FUNCTION_BLOCK "Epever_solar_charge_controller"   // FB109, SCL
{ S7_Optimized_Access := 'TRUE' }
VERSION : 0.1
   VAR_INPUT
      mb_addr : UInt := 1;
      on : Bool;
   END_VAR
   VAR_OUTPUT
      PV_array_input_voltage : Real;
      PV_array_input_current : Real;
      PV_array_input_power : Real;
      battery_power : Real;
      load_voltage : Real;
      load_current : Real;
      load_power : Real;
      battery_temperature : Real;
      temperature_inside_equipment : Real;
      battery_soc : Real;   // The percentage of battery's remaining capacity
      remote_battery_temperature : Real;
      battery_real_rated_power : Real;
      _ : Bool;
      PV_voltage_today_Maximum : Real;
      PV_voltage_today_Minimum : Real;
      Battery_voltage_today_Maximum : Real;
      Battery_voltage_today_Minimum : Real;
      Consumed_energy_today : Real;
      Consumed_energy_this_month : Real;
      Consumed_energy_this_year : Real;
      Consumed_energy_total : Real;
      Generated_energy_today : Real;
      Generated_energy_this_month : Real;
      Generated_energy_this_year : Real;
      Generated_energy_total : Real;
      Battery_voltage : Real;
      Battery_current : Real;
      __ : Bool;
      charging_status : Struct
         No_charging : Bool;
         Float : Bool;
         Boost : Bool;
         Equalization : Bool;
      END_STRUCT;
   END_VAR
   VAR_IN_OUT
      mb_query : "mb_query";
   END_VAR
   VAR
      sb : "mb_station_block_udt";
      read3 : Struct
         load_short : Bool;   // [08]
         load_over_current : Bool;   // [09]
         Input_is_over_current : Bool;   // [10]
         Anti_reverse_MOSFET_is_short : Bool;   // [11]
         Charging_or_Anti_reverse_MOSFET_is_short : Bool;   // [12]
         Charging_MOSFET_is_short : Bool;   // [13]
         x14 : Bool;   // [14]
         x15 : Bool;   // [15]
         Running : Bool;   // [00] - Standby
         Normal : Bool;   // [01] - Fault
         charging_status_0 : Bool;   // [02]
         charging_status_1 : Bool;   // [03]
         PV_Input_is_short : Bool;   // [04]
         x05 : Bool;   // [05]
         x06 : Bool;   // [06]
         Load_MOSFET_is_short : Bool;   // [07]
      END_STRUCT;
      first_scan : Bool := true;
   END_VAR
   VAR_TEMP
      read1 : Struct
         PV_array_input_voltage : UInt;   // [3100]
         PV_array_input_current : UInt;   // [3101]
         PV_array_input_power : UDInt;   // [3102]
         z_1 : Array[1..3] of Word;
         battery_power : UDInt;   // [3106]
         z_2 : Array[1..4] of Word;
         load_voltage : UInt;   // [310C]
         load_current : UInt;   // [310D]
         load_power : UDInt;   // [310E]
         battery_temperature : UInt;   // [3110]
         temperature_inside_equipment : UInt;   // [3111]
         battery_soc : UInt;   // [311A] The percentage of battery's remaining capacity
         remote_battery_temperature : UInt;   // [311B]
         z_3 : UInt;
         battery_real_rated_power : UInt;   // [311D]
      END_STRUCT;
      read2 : Struct
         PV_voltage_today_Maximum : UInt;   // [3300]
         PV_voltage_today_Minimum : UInt;   // [3301]
         Battery_voltage_today_Maximum : UInt;   // [3302]
         Battery_voltage_today_Minimum : UInt;   // [3303]
         Consumed_energy_today : UDInt;   // [3304]
         Consumed_energy_this_month : UDInt;   // [3306]
         Consumed_energy_this_year : UDInt;   // [3308]
         Consumed_energy_total : UDInt;   // [330A]
         Generated_energy_today : UDInt;   // [330C]
         Generated_energy_this_month : UDInt;   // [330E]
         Generated_energy_this_year : UDInt;   // [3310]
         Generated_energy_total : UDInt;   // [3312]
         Battery_voltage : UInt;   // [331A]
         Battery_current : UDInt;   // [331B]
      END_STRUCT;
      tmp : Byte;
   END_VAR
BEGIN
   // Epever - solar charge controller 
   // v2.3 - 12 june 2015
   // 

   IF #first_scan THEN
       #sb.conf.read_only := true;
   END_IF;

   "mb_station_block_header"(sb := #sb, mb_query := #mb_query);
   #mb_query.mb_addr := #mb_addr; 

   #mb_query.mode := #mb_query.c.read.input_reg;
   #mb_query(data_addr := 16#3100, data_ptr := #read1);
   IF #mb_query.Done THEN
       #PV_array_input_voltage := UINT_TO_REAL(#read1.PV_array_input_voltage) / 100;
       #PV_array_input_current := UINT_TO_REAL(#read1.PV_array_input_current) / 100;
       #PV_array_input_power := UDINT_TO_REAL(ROR(IN := #read1.PV_array_input_power, N := 16)) / 100;
       #battery_power := UDINT_TO_REAL(ROR(IN := #read1.battery_power, N := 16)) / 100;
       #load_voltage := UINT_TO_REAL(#read1.load_voltage) / 100;
       #load_current := UINT_TO_REAL(#read1.load_current) / 100;
       #load_power := UDINT_TO_REAL(ROR(IN := #read1.load_power, N := 16)) / 100;
       #battery_temperature := UINT_TO_REAL(#read1.battery_temperature) / 100;
       #temperature_inside_equipment := UINT_TO_REAL(#read1.temperature_inside_equipment) / 100;
       #battery_soc := UINT_TO_REAL(#read1.battery_soc) / 100;
       #remote_battery_temperature := UINT_TO_REAL(#read1.remote_battery_temperature) / 100;
       #battery_real_rated_power := UINT_TO_REAL(#read1.battery_real_rated_power) / 100;
   END_IF;

   #mb_query(data_addr := 16#3300, data_ptr := #read2);
   IF #mb_query.Done THEN
       #PV_voltage_today_Maximum := UINT_TO_REAL(#read2.PV_voltage_today_Maximum) / 100;
       #PV_voltage_today_Minimum := UINT_TO_REAL(#read2.PV_voltage_today_Minimum) / 100;
       #Battery_voltage_today_Maximum := UINT_TO_REAL(#read2.Battery_voltage_today_Maximum) / 100;
       #Battery_voltage_today_Minimum := UINT_TO_REAL(#read2.Battery_voltage_today_Minimum) / 100;
       #Consumed_energy_today := UDINT_TO_REAL(ROR(IN := #read2.Consumed_energy_today, N := 16)) / 100;
       #Consumed_energy_this_month := UDINT_TO_REAL(ROR(IN := #read2.Consumed_energy_this_month, N := 16)) / 100;
       #Consumed_energy_this_year := UDINT_TO_REAL(ROR(IN := #read2.Consumed_energy_this_year, N := 16)) / 100;
       #Consumed_energy_total := UDINT_TO_REAL(ROR(IN := #read2.Consumed_energy_total, N := 16)) / 100;
       #Generated_energy_today := UDINT_TO_REAL(ROR(IN := #read2.Generated_energy_today, N := 16)) / 100;
       #Generated_energy_this_month := UDINT_TO_REAL(ROR(IN := #read2.Generated_energy_this_month, N := 16)) / 100;
       #Generated_energy_this_year := UDINT_TO_REAL(ROR(IN := #read2.Generated_energy_this_year, N := 16)) / 100;
       #Generated_energy_total := UDINT_TO_REAL(ROR(IN := #read2.Generated_energy_total, N := 16)) / 100;
       #Battery_voltage := UDINT_TO_REAL(#read2.Battery_voltage) / 100;
       #Battery_current := UDINT_TO_REAL(ROR(IN := #read2.Battery_current, N := 16)) / 100;
   END_IF;


   #mb_query(data_addr := 16#3201, data_ptr := #read3);
   #tmp.%X0 := #read3.charging_status_0;
   #tmp.%X1 := #read3.charging_status_1;
   #charging_status.No_charging := #tmp = 0;
   #charging_status.Float := #tmp = 1;
   #charging_status.Boost := #tmp = 2;
   #charging_status.Equalization := #tmp = 3;

   #mb_query.mode := #mb_query.c.write.single_discrete_output;
   #tmp.%X0 := #on;
   #mb_query(data_addr := 0, data_ptr := #tmp);

   "mb_station_block_footer"(sb := #sb, mb_query := #mb_query);


   (*
   - 16bit MODBUS addresses (per the modbus.org spec)
   - BPS: 115200 baud
   - Parity: None
   - Data bits: 8
   - Stop bits: 1
   - Flow control: None

   Pin definition RJ45 
   1   Power supply output +7.5
   2   Power supply output +7.5
   3   RS-485 - A
   4   RS-485 - A
   5   RS-485 - B
   6   RS-485 - B
   7   Ground
   8   Ground

   *)
END_FUNCTION_BLOCK

// folder: Library/Modbus/Station blocks/sb Untested/F/Floridan

FUNCTION_BLOCK "Floridan_Uniflo_1200"   // FB83, SCL
{ S7_Optimized_Access := 'TRUE' }
VERSION : 0.1
   VAR_INPUT
      mb_addr : USInt;
      delay : Time := T#10S;
   END_VAR
   VAR_OUTPUT
      energi : LReal;   // [MJ]
      vol_measured : LReal;   // [m3]
      vol_conv : LReal;   // [Nm3]
      pressure : LReal;   // [bar A]
      temperature : LReal;
   END_VAR
   VAR_IN_OUT
      mb_query : "mb_query";
   END_VAR
   VAR
      sb : "mb_station_block_udt";
      battery_remaining : UInt;
      mb_delay : "mb_delay";
      serial_number : String[6];
   END_VAR
   VAR_TEMP
      dommy : Bool;
      c : Int;
      "dword" : DWord;
   END_VAR
BEGIN
   // Flonidan - Uniflo 1200 GVEC
   // Product number: 061864X-YYY
   //
   // - https://www.gavilar.nl/files/communicationboard230210_1521630740_b6a3b533.pdf
   // - M/06180XX/24

   "mb_station_block_header"(sb := #sb, mb_query := #mb_query);
   #mb_query.mb_addr := #mb_addr; // Device address.

   // Reduce power consumption, by halting execution. Nice if the device is running 
   // on battery. mb_delay is located inside the mb_extended_features.scl file.
   #mb_delay(delay := #delay, mb_query := #mb_query);

   #mb_query.mb_addr.%X5 := 0; // - Last bits of mb_addr is used for expanding 
   #mb_query.mb_addr.%X6 := 0; //   register addr, this means that only addr 1
   #mb_query.mb_addr.%X7 := 0; //   to 31 on the bus may be used.

   #mb_query.mode := #mb_query.c.read.holding_reg;

   #mb_query(data_addr := 123, data_ptr := #battery_remaining);
   #mb_query(data_addr := 2833, data_ptr := #serial_number); // Serial number 

   #mb_query.conf.buffer_handler := false;

   #mb_query(data_addr := 56, data_len := 44, data_ptr := #dommy);
   IF #mb_query.Done THEN
       #vol_conv := "intreal"(mb_query := #mb_query, addr := 16#70 / 2);
       #"dword".%B3 := #mb_query.z.buffer[16]; // 16#80/2=64, (64-56)*2=16
       #"dword".%B2 := #mb_query.z.buffer[17];
       #"dword".%B1 := #mb_query.z.buffer[18];
       #"dword".%B0 := #mb_query.z.buffer[19];
       #pressure := DWORD_TO_REAL(#"dword");
       #"dword".%B3 := #mb_query.z.buffer[20]; // 16#84/2=66, (66-56)*2=20
       #"dword".%B2 := #mb_query.z.buffer[21];
       #"dword".%B1 := #mb_query.z.buffer[22];
       #"dword".%B0 := #mb_query.z.buffer[23];
       #temperature := DWORD_TO_REAL(#"dword");
       #energi := "intreal"(mb_query := #mb_query, addr := 16#90 / 2);
       #vol_measured := "intreal"(mb_query := #mb_query, addr := 16#98 / 2);
   END_IF;

   #mb_query.data_len := #mb_query.c.auto_len;
   #mb_query.conf.buffer_handler := true;
   "mb_station_block_footer"(sb := #sb, mb_query := #mb_query);
END_FUNCTION_BLOCK

FUNCTION "intreal" : LReal   // FC16, SCL
{ S7_Optimized_Access := 'TRUE' }
VERSION : 0.1
   VAR_INPUT
      mb_query : "mb_query";
      addr : UInt;
   END_VAR
   VAR_TEMP
      dw : UDInt;
      r : DWord;
      bo : UDInt;
   END_VAR
BEGIN
   // Uniflo 1200 has a special datatype named
   // int-real, this block decode that data type.

   // buffer offset
   #bo := (#addr - #mb_query.data_addr) * 2;

   // The integer part of the value, little endian.
   #dw.%B3 := #mb_query.z.buffer[#bo + 0];
   #dw.%B2 := #mb_query.z.buffer[#bo + 1];
   #dw.%B1 := #mb_query.z.buffer[#bo + 2];
   #dw.%B0 := #mb_query.z.buffer[#bo + 3];
   #intreal := UDINT_TO_LREAL(#dw);

   // The decimal part of the value, little endian.
   // Stored as a real (IEEE754).
   #r.%B3 := #mb_query.z.buffer[#bo + 4];
   #r.%B2 := #mb_query.z.buffer[#bo + 5];
   #r.%B1 := #mb_query.z.buffer[#bo + 6];
   #r.%B0 := #mb_query.z.buffer[#bo + 7];
   #intreal += DWORD_TO_REAL(#r);
END_FUNCTION

// folder: Library/Modbus/Station blocks/sb Untested/G

FUNCTION_BLOCK "G_Instruments_GpH141_MB"   // FB26, SCL
{ S7_Optimized_Access := 'TRUE' }
VERSION : 0.1
   VAR_INPUT
      mb_addr : USInt;
   END_VAR
   VAR_OUTPUT
      voltage_mV : Real;
      pH : Real;
      temperature : Real;
   END_VAR
   VAR_IN_OUT
      mb_query : "mb_query";
   END_VAR
   VAR
      sb : "mb_station_block_udt";
      change_mb_addr : Struct
         old : UInt;
         new : UInt;
      END_STRUCT;
   END_VAR
   VAR_TEMP
      read1 : Struct
         voltage : Int;
         pH : Int;   // compensated for temperature
         temperature : Int;
      END_STRUCT;
   END_VAR
BEGIN
   // G Instruments - GpH141-MB - pH/ORP Transmitter
   // Part number: 30535.
   // http://www.ginstruments.com/files/GpH141-MB.pdf

   "mb_station_block_header"(sb := #sb, mb_query := #mb_query);
   #mb_query.mb_addr := #mb_addr;

   #mb_query.mode := #mb_query.c.read.holding_reg;

   #mb_query(data_addr := 19, data_ptr := #read1);
   IF #mb_query.Done THEN
       #voltage_mV := INT_TO_REAL(#read1.voltage) / 10;
       #pH := INT_TO_REAL(#read1.pH) / 100;
       #temperature := INT_TO_REAL(#read1.temperature) / 10;
   END_IF;

   (* IF #change_mb_addr.new <> 0 AND #change_mb_addr.old <> 0 THEN
       #mb_query(mb_addr := #change_mb_addr.old,
                 mode := #mb_query.c.write.single_holding_reg,
                 data_addr := 1200,
                 data_ptr := #change_mb_addr.new);
       IF #mb_query.Done THEN #change_mb_addr.new := 0; END_IF;
   END_IF; *)

   "mb_station_block_footer"(sb := #sb, mb_query := #mb_query);

   (*
   Default comm. setting: 19200 bps, even parity, addr 1.

   Electrical connection:
   10 is A (D+)
   11 is RS485 ground (isolated from all other grounds)
   12 is B (D-)
   *)
END_FUNCTION_BLOCK

// folder: Library/Modbus/Station blocks/sb Untested/G/Grundfoss

FUNCTION_BLOCK "Grunnfoss_pump"   // FB14, SCL
{ S7_Optimized_Access := 'TRUE' }
VERSION : 0.1
   VAR_INPUT
      mb_addr : USInt;
      setpoint : Real;   // [%]
   END_VAR
   VAR_OUTPUT
      ProcessFeedback : Real;
      _ : Bool;
      Head : Real;   // bar
      VolumeFlow : Real;   // m3/h
      RelativePerformance : Real;   // %
      Speed : Real;   // rpm
      Frequency : Real;   // Hz
      ActualSetpoint : Real;   // %
      MotorCurrent : Real;   // A
      DCLinkVoltage : Real;   // V
      MotorVoltage : Real;   // V
      Power : Real;   // W
      RemoteFlow : Real;   // m3/h
      InletPressure : Real;   // bar
      RemotePressure : Real;   // bar
      Level : Real;   // m
      PowerElectronicTemp : Real;   // degree C
      MotorTemp : Real;   // degree C
      RemoteTemp : Real;   // degree C
      ElectronicTemp : Real;   // degree C
      PumpLiquidTemp : Real;   // degree C
      BearingTempDE : Real;   // degree C
      BearingTempNDE : Real;   // degree C
      AuxSensorInput : Real;   // %
      SpecificEnergyConsumption : Real;   // Wh/m3
      OperationTime : Real;   // hour
      TotalPoweredTime : Real;   // hour
      Torque : Real;   // Nm
      Energy : Real;   // kWh
      NumberOfStarts : Real;
   END_VAR
   VAR_IN_OUT
      mb_query : "mb_query";
   END_VAR
   VAR
      sb : "mb_station_block_udt";
      read1 : Struct
         status : Struct   // (201)
            x08_AccessModeRemote : Bool;
            x09_On : Bool;
            x10_Fault : Bool;
            x11_Warning : Bool;
            x12_ForcedToLocal : Bool;
            x13_AtMaxSpeed : Bool;
            x14 : Bool;
            x15_AtMinSpeed : Bool;
            x00_LowFlowStop : Bool;
            x01_CopyToLocal : Bool;
            x02_MaxFlowLimitEnabled : Bool;
            x03_ResetAlarmAck : Bool;
            x04_SetpointInfluence : Bool;
            x05_AtMaxPower : Bool;
            x06_Rotation : Bool;
            x07_Direction : Bool;
         END_STRUCT;
         ProcessFeedback : UInt;   // (202) x 0.01
         ControlMode : UInt;   // (203)
         OperationMode : UInt;   // (204)
         AlarmCode : UInt;   // (205)
         WarningCode : UInt;   // (206)
         MonthsToBearingService : Byte;   // (207)
         BearingServiceType : Byte;
         DriveState : UInt;   // (208)
         FeedbackSensorUnit : UInt;   // (209)
         FeedbackSensorMin : UInt;   // (210)
         FeedbackSensorMax : UInt;   // (211)
         NominalFrequency : UInt;   // (212)
         MinFrequency : UInt;   // (213) Minimum frequency in % of nominal frequency
         MaxFrequency : UInt;   // (214) Maximum frequency in % of nominal frequency
         SetpointRangeMin : UInt;   // (215)
         SetpointRangeMax : UInt;   // (216)
         _ : Array[1..4] of UInt;
         FlowEstimationState : UInt;   // (221) 0: within range, 1:below, 2:above
      END_STRUCT;
      read2 : Struct
         Head : UInt;   // (301) 0.001 bar
         VolumeFlow : UInt;   // (302) 0.1 m3/h
         RelativePerformance : UInt;   // (303) 0.01 %
         Speed : UInt;   // (304) rpm
         Frequency : UInt;   // (305) 0.1 Hz
         DigitalInput : Word;   // (306)
         DigitalOutput : Word;   // (307)
         ActualSetpoint : UInt;   // (308) 0.01 %
         MotorCurrent : UInt;   // (309) 0.1 A
         DCLinkVoltage : UInt;   // (310) 0.1 V
         MotorVoltage : UInt;   // (311) 0.1 V
         Power : UDInt;   // (312) W
         RemoteFlow : UInt;   // (314) 0.1 m3/h
         InletPressure : UInt;   // (315) 0.001 bar
         RemotePressure : UInt;   // (316) 0.001 bar
         Level : UInt;   // (317) 0.01 m
         PowerElectronicTemp : UInt;   // (318) 0.01 K
         MotorTemp : UInt;   // (319) 0.01 K
         RemoteTemp : UInt;   // (320) 0.01 K
         ElectronicTemp : UInt;   // (321) 0.01 K
         PumpLiquidTemp : UInt;   // (322) 0.01 K
         BearingTempDE : UInt;   // (323) 0.01 K
         BearingTempNDE : UInt;   // (324) 0.01 K
         AuxSensorInput : UInt;   // (325) 0.01 %
         SpecificEnergyConsumption : UInt;   // (326) Wh/m3
         OperationTime : UDInt;   // (327) hour
         TotalPoweredTime : UDInt;   // (329) hour
         Torque : UInt;   // (331) 0.1 Nm
         Energy : UDInt;   // (332) kWh
         NumberOfStarts : UDInt;   // (334)
      END_STRUCT;
      write : Struct
         cmd : Struct   // (101)
            x08 : Bool;
            x09 : Bool;
            x10 : Bool;
            x11 : Bool;
            x12 : Bool;
            x13 : Bool;
            x14 : Bool;
            x15 : Bool;
            x00_Remote : Bool := true;   // 0=Local
            x01_On : Bool;   // 0=Off
            x02_ResetAlarm : Bool;   // rising edge only
            x03_CopyToLocal : Bool;
            x04_EnableMaxFlowLimit : Bool;
            x05 : Bool;
            x06 : Bool;
            x07 : Bool;
         END_STRUCT;
         ControlMode : UInt;   // (102)
         OperationMode : UInt;   // (103)
         Setpoint : UInt;   // (104)
         Relay : Struct   // (105)
            x08 : Bool;
            x09 : Bool;
            x10 : Bool;
            x11 : Bool;
            x12 : Bool;
            x13 : Bool;
            x14 : Bool;
            x15 : Bool;
            x00_Realy1_inverted : Bool;   // 0: Closed, 1:Open
            x01_Realy2_inverted : Bool;   // 0: Closed, 1:Open
            x02_Realy3_inverted : Bool;   // 0: Closed, 1:Open
            x03_Realy4_inverted : Bool;   // 0: Closed, 1:Open
            x04 : Bool;
            x05 : Bool;
            x06 : Bool;
            x07 : Bool;
            x : Struct
               x08 : Bool;
               x09 : Bool;
               x10 : Bool;
               x11 : Bool;
               x12 : Bool;
               x13 : Bool;
               x14 : Bool;
               x15 : Bool;
               x00 : Bool;
               x01 : Bool;
               x02 : Bool;
               x03 : Bool;
               x04 : Bool;
               x05 : Bool;
               x06 : Bool;
               x07 : Bool;
            END_STRUCT;
            x_1 : Struct
               x08 : Bool;
               x09 : Bool;
               x10 : Bool;
               x11 : Bool;
               x12 : Bool;
               x13 : Bool;
               x14 : Bool;
               x15 : Bool;
               x00 : Bool;
               x01 : Bool;
               x02 : Bool;
               x03 : Bool;
               x04 : Bool;
               x05 : Bool;
               x06 : Bool;
               x07 : Bool;
               x : Struct
                  x08 : Bool;
                  x09 : Bool;
                  x10 : Bool;
                  x11 : Bool;
                  x12 : Bool;
                  x13 : Bool;
                  x14 : Bool;
                  x15 : Bool;
                  x00 : Bool;
                  x01 : Bool;
                  x02 : Bool;
                  x03 : Bool;
                  x04 : Bool;
                  x05 : Bool;
                  x06 : Bool;
                  x07 : Bool;
               END_STRUCT;
            END_STRUCT;
         END_STRUCT;
         SetMaxFlowLimit : UInt;   // (106) 0.01 m3/h
      END_STRUCT;
   END_VAR
BEGIN
   // Grundfoss - Pumps
   // CIM 200 Modbus RTU
   // CIM 500 Modbus TCP

   "mb_station_block_header"(sb := #sb, mb_query := #mb_query);
   #mb_query.mb_addr := #mb_addr;

   #mb_query.mode := #mb_query.c.read.holding_reg;

   #mb_query(data_addr := 201, data_ptr := #read1);
   IF #mb_query.Done THEN
       #ProcessFeedback := UINT_TO_REAL(#read1.ProcessFeedback) / 100;
   END_IF;

   #mb_query(data_addr := 301, data_ptr := #read2);
   IF #mb_query.Done THEN
       #Head := UINT_TO_REAL(#read2.Head) * 0.001;
       #VolumeFlow := UINT_TO_REAL(#read2.VolumeFlow) * 0.1;
       #RelativePerformance := UINT_TO_REAL(#read2.RelativePerformance) * 0.01;
       #Speed := UINT_TO_REAL(#read2.Speed);
       #Frequency := UINT_TO_REAL(#read2.Frequency) * 0.1;
       #ActualSetpoint := UINT_TO_REAL(#read2.ActualSetpoint) * 0.01;
       #MotorCurrent := UINT_TO_REAL(#read2.MotorCurrent) * 0.1;
       #DCLinkVoltage := UINT_TO_REAL(#read2.DCLinkVoltage) * 0.1;
       #MotorVoltage := UINT_TO_REAL(#read2.MotorVoltage) * 0.1;
       #Power := UDINT_TO_REAL(#read2.Power);
       #RemoteFlow := UINT_TO_REAL(#read2.RemoteFlow) * 0.1;
       #InletPressure := UINT_TO_REAL(#read2.InletPressure) * 0.001;
       #RemotePressure := UINT_TO_REAL(#read2.RemotePressure) * 0.001;
       #Level := UINT_TO_REAL(#read2.Level) * 0.01;
       #PowerElectronicTemp := UINT_TO_REAL(#read2.PowerElectronicTemp) * 0.01 - 273.15;
       #MotorTemp := UINT_TO_REAL(#read2.MotorTemp) * 0.01 - 273.15;
       #RemoteTemp := UINT_TO_REAL(#read2.RemoteTemp) * 0.01 - 273.15;
       #ElectronicTemp := UINT_TO_REAL(#read2.ElectronicTemp) * 0.01 - 273.15;
       #PumpLiquidTemp := UINT_TO_REAL(#read2.PumpLiquidTemp) * 0.01 - 273.15;
       #BearingTempDE := UINT_TO_REAL(#read2.BearingTempDE) * 0.01 - 273.15;
       #BearingTempNDE := UINT_TO_REAL(#read2.BearingTempNDE) * 0.01 - 273.15;
       #AuxSensorInput := UINT_TO_REAL(#read2.AuxSensorInput) * 0.01;
       #SpecificEnergyConsumption := UINT_TO_REAL(#read2.SpecificEnergyConsumption);
       #OperationTime := UDINT_TO_REAL(#read2.OperationTime);
       #TotalPoweredTime := UDINT_TO_REAL(#read2.TotalPoweredTime);
       #Torque := UINT_TO_REAL(#read2.Torque) * 0.1;
       #Energy := UDINT_TO_REAL(#read2.Energy);
       #NumberOfStarts := UDINT_TO_REAL(#read2.NumberOfStarts);
   END_IF;


   // Write preparations
   #write.cmd.x01_On := #setpoint <> 0;
   #write.Setpoint := REAL_TO_UINT(#setpoint * 100);

   #mb_query.mode := #mb_query.c.write.holding_reg;
   #mb_query(data_addr := 101, data_ptr := #write);

   "mb_station_block_footer"(sb := #sb, mb_query := #mb_query);

   (*

   #write.ControlMode:
   Some modes are not supported by all E-pumps.
   0: Constant speed
   1: Constant frequency
   3: Constant head
   4: Constant pressure
   5: Constant differential pressure
   6: Proportional pressure
   7: Constant flow
   8: Constant temperature
   10: Constant level
   128: AUTOADAPT
   129: FLOWADAPT (set FLOWLIMIT in register 00106)
   130: Closed-loop sensor.

   #write.OperationMode:
   0: Auto-control (setpoint control according to selected control mode)
   4: OpenLoopMin (running at minimum speed)
   6: OpenLoopMax (running at maximum speed)

   #read.DriveState:
   0: Stopped
   1: Accelerating
   2: Decelerating
   3: Steady state/closed loop
   4: -
   5: Accelerating halt
   6: Decelerating halt
   7: Start on the run (flying cut-in)
   Only MGE motors and CUE drives.

   #read.FeedbackSensorUnit:
   0: bar
   1: mbar
   2: m
   3: kPa
   4: psi
   5: ft
   6: m3/h
   7: m3/s
   8: l/s
   9: gpm
   10: °C
   11: °F
   12: %
   13: K
   14: W

   *)
END_FUNCTION_BLOCK

// folder: Library/Modbus/Station blocks/sb Untested/H

FUNCTION_BLOCK "Hitachi_wj200_series"   // FB27, SCL
{ S7_Optimized_Access := 'TRUE' }
VERSION : 0.1
   VAR_INPUT
      mb_addr : USInt;
      ref : Real;
      acceleration_time : Real := 30.0;   // sec
      deceleration_time : Real := 30.0;   // sec
   END_VAR
   VAR_OUTPUT
      output_frequency : Real;
      output_current : Real;
   END_VAR
   VAR_IN_OUT
      mb_query : "mb_query";
   END_VAR
   VAR
      sb : "mb_station_block_udt";
      save_param : Bool;
      read1 : Struct
         output_frequency : UDInt;   // 0.01 [Hz]
         output_current : UInt;   // 0.1 [A]
         rotation_direction : Int;   // 0: Stopping, 1: Forward, 2:Reverse
      END_STRUCT;
      read2 : Struct
         torque : Int;   // [%]
         output_voltage : UInt;   // 0.1 [V]
         output_power : UInt;   // 0.1 [kW]
         watt_hour : UDInt;   // 0.1 [wh]
         elapsed_run_time : UDInt;   // [h]
         elapsed_power_on_time : UDInt;   // [h]
         "heat sink_temperature" : UDInt;   // 0.1 [℃]
      END_STRUCT;
      read3_Life_check : Struct
         x08 : Bool;
         x09 : Bool;
         x10 : Bool;
         x11 : Bool;
         x12 : Bool;
         x13 : Bool;
         x14 : Bool;
         x15 : Bool;
         x00_Capacitor_on_main_circuit_board : Bool;
         x01_cooling_fan : Bool;
         x02 : Bool;
         x03 : Bool;
         x04 : Bool;
         x05 : Bool;
         x06 : Bool;
         x07 : Bool;
      END_STRUCT;
      read4_Ambient_temperature : Int;
      read5_trip : Struct
         cnt : UInt;
         info : Array[1..3] of Struct
            factor : UInt;
            status : UInt;
            frequency : DInt;
            current : UInt;
            voltage : UInt;
            running_time : UDInt;   // [h] Cumulative running time at tripping
            powerOn_time : UDInt;   // [h] Cumulative power-on time at tripping
         END_STRUCT;
      END_STRUCT;
      read6_status : Struct
         "A" : UInt;
         "B" : UInt;   // 0: Stopping, 1: Running, 2: Tripping
         C : UInt;
      END_STRUCT;
      read7 : Struct
         x0_inverter_ready : Bool;
         x1_forward : Bool;
         x2_reverse : Bool;
         x3_major_failure : Bool;
         x4_data_writing_in_progress : Bool;
         x5 : Bool;
         x6 : Bool;
         x7 : Bool;
      END_STRUCT;
      write1 : Struct
         acceleration_time_1 : UDInt := 3000;   // x0.01 sec
         deceleration_time_1 : UDInt := 3000;   // x0.01 sec
      END_STRUCT;
      write2_source : Struct
         frequency_source : UInt := 3;   // 3:Modbus
         run_command_source : UInt := 3;   // 3:Modbus
      END_STRUCT;
      write3_comm_error : Struct
         communication_watchdog_timer : UInt := 1000;   // 0.01 [sec.]
         communication_error_action : UInt := 4;
      END_STRUCT;
      write5 : Struct
         x0_Run : Bool;
         x1_Reverse : Bool;
         x2_Trip : Bool;
         x3_Reset : Bool;
         x4 : Bool;
         x5 : Bool;
         x6 : Bool;
         x7 : Bool;
      END_STRUCT;
      write6_DC_breaking : Struct
         enable : UInt;   // 0 (disabling), 1 (enabling), 2 (output freq < [A052])
         frequency : UInt;   // 0.01 [Hz]
         wait_time : UInt;   // 0.1 [sec.]
         force_during_deceleration : UInt;   // [%]
         time_for_deceleration : UInt;   // 0.1 [sec.]
      END_STRUCT;
   END_VAR
   VAR_TEMP
      tmp : Word;
      write4_frequency : DInt;   // 0.01 [Hz]
   END_VAR
BEGIN
   // Hitachi WJ200-series
   // Manual Number: NT325X
   // https://www.hitachi-america.us/supportingdocs/forbus/inverters/Support/WJ200_Instruction_NT325X.pdf

   "mb_station_block_header"(sb := #sb, mb_query := #mb_query);
   #mb_query.mb_addr := #mb_addr;

   // --- Read queries
   #mb_query.mode := #mb_query.c.read.holding_reg;
   #mb_query(data_addr := 16#1001, data_ptr := #read1);
   #mb_query(data_addr := 16#1010, data_ptr := #read2);
   #mb_query(data_addr := 16#101d, data_ptr := #read3_Life_check);
   #mb_query(data_addr := 16#134e, data_ptr := #read4_Ambient_temperature);
   #mb_query(data_addr := 16#0011, data_ptr := #read5_trip);
   #mb_query(data_addr := 16#0003, data_ptr := #read6_status);

   #output_frequency := UDINT_TO_REAL(#read1.output_frequency) / 100;
   #output_current := UINT_TO_REAL(#read1.output_current) / 10;

   #mb_query(mode := #mb_query.c.read.discrete_output,
             data_addr := 16#0045,
             data_ptr := #read7);

   // --- Write queries ---
   #write4_frequency := REAL_TO_DINT(#ref * 100);
   #write1.acceleration_time_1 := REAL_TO_UDINT(#acceleration_time * 100);
   #write1.deceleration_time_1 := REAL_TO_UDINT(#deceleration_time * 100);

   #mb_query.mode := #mb_query.c.write.holding_reg;
   #mb_query(data_addr := 16#1103, data_ptr := #write1);
   #mb_query(data_addr := 16#1201, data_ptr := #write2_source);
   #mb_query(data_addr := 16#162e, data_ptr := #write3_comm_error);
   #mb_query(data_addr := 16#0001, data_ptr := #write4_frequency);
   #mb_query(data_addr := 16#1245, data_ptr := #write6_DC_breaking);

   // Save data to EEPROM. 
   IF #save_param THEN
       #mb_query(mode := #mb_query.c.write.single_holding_reg,
                 data_addr := 16#0900,
                 data_ptr := #tmp);
       #save_param := NOT #mb_query.Done;
   END_IF;

   #write5.x0_Run := #ref <> 0;
   #mb_query(mode := #mb_query.c.write.discrete_output,
             data_addr := 16#0001,
             data_len := 4,
             data_ptr := #write5);

   #mb_query.data_len := #mb_query.c.auto_len;
   "mb_station_block_footer"(sb := #sb, mb_query := #mb_query);

   (*
   === read6_status ===
   .A
   0: Initial status
   2: Stopping
   3: Running
   4: Free-run stop
   5: Jogging
   6: DC braking
   7: Retrying
   8: Tripping
   9: Undervoltage (UV), 

   .C
   1: Stopping
   2: Decelerating
   3: Constant-speed operation
   4: Accelerating
   5: Forward rotation
   6: Reverse rotation
   7: Switching from fwd. to rev. rotation,
   8: Switching from rev. to fwd. rotation,
   9: Starting fwd.
   10: Starting rev

   === write3_comm_error.communication_error_action === 
   0 (tripping), 
   1 (tripping after decelerating and stopping the motor), 
   2 (ignoring errors),
   3 (stopping the motor after free-running),
   4 (decelerating and stopping the motor) 

   === Save data to EEPROM === 
   The service life of the storage element of the inverter is 
   limited to about 100,000 write operations.  Frequent use of 
   the ENTER command may shorten its service life.

   === read5_trip.info ===
   .factor: 
   00 No trip factor 0 
   01 Over-current event while at constant speed 1 
   02 Over-current event during deceleration 2 
   03 Over-current event during acceleration 3 
   04 Over-current event during other conditions 4 
   05 Overload protection 5 
   06 Braking resistor overload protection 6 
   07 Overvoltage protection 7 
   08 EEPROM error 8 
   09 Undervoltage protection 9
   10 Current detection error 10
   11 CPU error 11
   12 External trip 12
   13 USP error 13
   14 Ground-fault protection 14
   15 Input overvoltage protection 15
   21 Inverter thermal trip 21
   22 CPU error 22
   25 Main circuit error 25
   30 Driver error 30
   35 Thermistor error 35
   36 Braking error 36
   37 Safe Stop 37
   38 Low-speed overload protection 38
   40 Operator connection 40
   41 Modbus communication error 41
   43 Easy sequence error (invalid instruction) 43
   44 Easy sequence error (invalid nesting count) 44
   45 Easy sequence execution error 1 45
   50 Easy sequence user trip 0 to 9, 50 to 59
   60 Option error 0 to 9, 60 to 69
   80 Encoder disconnection 80
   81 Excessive speed 81
   83 Position control range trip 83

   .status
   0: Resetting 
   1: Stopping 
   2: Decelerating 
   3: Constant-speed operation 
   4: Accelerating 
   5: Operating at zero frequency 
   6: Starting 
   7: DC braking 
   8: Overload restricted 

   *)
END_FUNCTION_BLOCK

// folder: Library/Modbus/Station blocks/sb Untested/H/Honeywell

FUNCTION_BLOCK "Honeywell_UDA2182"   // FB28, SCL
{ S7_Optimized_Access := 'TRUE' }
VERSION : 0.1
   VAR_INPUT
      mb_addr : UInt;
   END_VAR
   VAR_IN_OUT
      mb_query : "mb_query";
   END_VAR
   VAR
      sb : "mb_station_block_udt";
      data : Struct
         pv1 : Array[1..2] of Real;
         temperature : Array[1..2] of Real;
         alarm : Array[1..4] of DWord;
      END_STRUCT;
   END_VAR
BEGIN
   // Honeywell - UDA2182
   // 
   // Web: https://www.honeywellprocess.com/library/support/Public/Documents/70-82-25-126.pdf

   "mb_station_block_header"(sb := #sb, mb_query := #mb_query);
   #mb_query.mb_addr := #mb_addr;

   #mb_query.mode := #mb_query.c.mode.read;
   #mb_query(data_addr := 30001, data_ptr := #data);

   "mb_station_block_footer"(sb := #sb, mb_query := #mb_query);
END_FUNCTION_BLOCK

FUNCTION_BLOCK "Honeywell_variable_frequency_drives"   // FB29, SCL
{ S7_Optimized_Access := 'TRUE' }
VERSION : 0.1
   VAR_INPUT
      mb_addr : UInt := 255;
   END_VAR
   VAR_IN_OUT
      mb_query : "mb_query";
   END_VAR
   VAR
      sb : "mb_station_block_udt";
      read : Struct
         stw : Struct
            x24 : Bool;
            x25 : Bool;
            x26 : Bool;
            x27 : Bool;
            x28 : Bool;
            x29_control_place : Bool := FALSE;
            x30_control_place : Bool := FALSE;
            x31_control_place : Bool := TRUE;
            x16 : Bool;
            x17 : Bool;
            x18 : Bool;
            x19 : Bool;
            x20 : Bool;
            x21 : Bool;
            x22 : Bool;
            x23 : Bool;
            x08 : Bool;
            x09 : Bool;
            x10 : Bool;
            x11 : Bool;
            x12 : Bool;
            x13 : Bool;
            x14 : Bool;
            x15 : Bool;
            x00_Ready : Bool;
            x01_Running : Bool;
            x02_Counterclockwise : Bool;
            x03_Faulted : Bool;
            x04_Alarm : Bool;
            x05_AtReference : Bool;
            x06_ZeroSpeed : Bool;
            x07_FluxReady : Bool;
         END_STRUCT;
         d1_Output_Frequency : DInt;   // 0,01 Hz
         d2_Motor_Speed : DInt;   // 1 rpm
         d3_Motor_Current : DInt;   // 0,1 A
         d4_Motor_Torque : DInt;   // 0,1 %
         d5_Motor_Power : DInt;   // 0,1 %
         d6_Motor_Voltage : DInt;   // 0,1 V
         d7_DC_link_voltage : DInt;   // 1 V
         d8_Active_Fault_Code : DInt;
      END_STRUCT;
      write : Struct
         ctw : Struct
            x08 : Bool;
            x09 : Bool;
            x10 : Bool;
            x11 : Bool;
            x12 : Bool;
            x13 : Bool;
            x14 : Bool;
            x15 : Bool;
            x00 : Bool;
            x01_start : Bool := TRUE;
            x02_Reverse : Bool;
            x03_Reset_faults : Bool;
            x04 : Bool;
            x05 : Bool;
            x06 : Bool;
            x07 : Bool;
         END_STRUCT;
         __ : Word;
         speed_ref : UInt;   // 0â€¦10000 %
      END_STRUCT;
   END_VAR
BEGIN
   // Honeywell - Variable frequency drives
   // 
   // Web: https://customer.honeywell.com/resources/techlit/
   //      TechLitDocuments/62-0000s/62-0351.pdf

   "mb_station_block_header"(sb := #sb, mb_query := #mb_query);
   #mb_query.mb_addr := #mb_addr;

   #mb_query(mode := #mb_query.c.read.holding_reg,
             data_addr := 2151,
             data_ptr := #read);

   #mb_query(mode := #mb_query.c.write.holding_reg,
             data_addr := 2001,
             data_ptr := #write);

   "mb_station_block_footer"(sb := #sb, mb_query := #mb_query);
END_FUNCTION_BLOCK

// folder: Library/Modbus/Station blocks/sb Untested/I

FUNCTION_BLOCK "InSitu_RDO_PRO_X"   // FB30, SCL
{ S7_Optimized_Access := 'TRUE' }
VERSION : 0.1
   VAR_INPUT
      mb_addr : UInt;
   END_VAR
   VAR_OUTPUT
      dissolved_oxygen : Real;   // mg/L
      temperature : Real;   // C
      saturation : Real;   // %
      oxygen_partial_pressure : Real;   // mbar
      alarm : Bool;
   END_VAR
   VAR_IN_OUT
      mb_query : "mb_query";
   END_VAR
   VAR
      sb : "mb_station_block_udt";
      read1 : Array[1..4] of Struct
         value : Real;
         Parameter_ID : UInt;
         Units_ID : UInt;
         data_quality : UInt;
         "Off line_sentinel_value" : UInt;
         Available_Units : UInt;
      END_STRUCT;
      read2 : Struct
         serial_number : UDInt;
         manufacture_date : Array[1..3] of UInt;
      END_STRUCT;
      device_name : String[32];
   END_VAR
   VAR_TEMP
      tmp_alarm : Bool;
      c : Int;
   END_VAR
BEGIN
   // InSitu - RDO PRO X
   // 
   // https://in-situ.com/wp-content/uploads/2015/08/
   // RDO_PRO-X_-Titan_Modbus_SDI-12-_Guide.pdf

   "mb_station_block_header"(sb := #sb, mb_query := #mb_query);
   #mb_query.mb_addr := #mb_addr;

   #mb_query.mode := #mb_query.c.read.holding_reg;
   #mb_query(data_addr := 38, data_ptr := #read1);
   #mb_query(data_addr := 9002, data_ptr := #read2);
   #mb_query(data_addr := 9019, data_ptr := #device_name);

   #dissolved_oxygen := #read1[1].value;
   #temperature := #read1[2].value;
   #saturation := #read1[3].value;
   #oxygen_partial_pressure := #read1[4].value;
   FOR #c := 1 TO 4 DO
       #tmp_alarm := #tmp_alarm OR #read1[#c].data_quality <> 0;
   END_FOR;
   #alarm := #tmp_alarm;

   "mb_station_block_footer"(sb := #sb, mb_query := #mb_query);

   (* 
   === Sensor health table: ===
   0  Normal Data Quality
   1  Parameter measured without errors using an expired user 
      calibration. (User Cal Expired)
   2  Parameter measured without errors using an expired factory 
      calibration. (Factory Cal Expired)
   3  Parameter measured with error, sentinel value supplied. 
   4  Sensor is warming up, sentinel value supplied.
   5  Parameter measured but does not meet normal quality 
      criteria. The sensor has sustained moderate damage, or  
      the recommended lifespan has been reached.
   *)
END_FUNCTION_BLOCK

FUNCTION_BLOCK "Integron_OXY-DIOS-DSP"   // FB84, SCL
{ S7_Optimized_Access := 'TRUE' }
VERSION : 0.1
   VAR_INPUT
      mb_addr : USInt;
   END_VAR
   VAR_IN_OUT
      mb_query : "mb_query";
   END_VAR
   VAR
      sb : "mb_station_block_udt";
      read1 : Struct
         Sensor_status : Struct
            x08 : Bool;
            x09 : Bool;
            x10 : Bool;
            x11 : Bool;
            x12 : Bool;
            x13 : Bool;
            x14 : Bool;
            x15 : Bool;
            x00_Correct_indication : Bool;
            x01_Range_exceeded_error : Bool;
            x02_Measuring_window_status : Bool;   // (Must be replaced)
            x03_Cleaning : Bool;
            x04_Maintaining_values_after_cleaning : Bool;   // ("holding time") F= Real current value, T=Saved value
            x05_Output_short_circuit_OXYGEN_CONTROL : Bool;
            x06_Output_short_circuit_AIRBLAST_CLEANING : Bool;
            x07 : Bool;
         END_STRUCT;
         cO2_concentration : Real;   // [mg/L]
         sO2_saturation : Real;   // [%]
         Head_temperature : Real;   // [degree C]
         pO2_O2_partial_pressure : Real;   // [bar]
         Tau_fluorescence_decay_time : Real;   // [us]
         Atmospheric_pressure : Real;   // [bar] (hydrostatic)
         Relative_humidity_inside_the_sensor : Real;   // [%]
         Humidity_sensor_temperature : Real;   // [degree C]
         Salinity : Real;   // [ppt]
         Mainboard_temperature : Real;   // [degree C]
         Sensor_serial_number : Array[1..4] of Word;
         Date_and_time : UDInt;   // [s]
         Window_serial_number : UInt;
         Expected_date_of_exchange_measuring_window : UDInt;   // [s]
         Date_of_last_calibration : UDInt;   // [s]
         RTC_battery_level : UInt;   // [%]
         Supply_power_24V : Real;
      END_STRUCT;
   END_VAR
BEGIN
   // Integron Poland EU - OXY-DIOS-DSP
   // Optical dissolved oxygen sensor
   // 
   // https://www.tme.eu/en/Document/9d0bf7a4d6041739cc6d58df1cc838cb/OXY-DIOS-DSP-Manual-EN-v.1.33.pdf
   // http://www.sensor.integron.pl

   "mb_station_block_header"(sb := #sb, mb_query := #mb_query);
   #mb_query.mb_addr := #mb_addr;

   #mb_query.mode := #mb_query.c.mode.read;
   #mb_query(data_addr := 41000, data_ptr := #read1);

   "mb_station_block_footer"(sb := #sb, mb_query := #mb_query);
END_FUNCTION_BLOCK

// folder: Library/Modbus/Station blocks/sb Untested/J

FUNCTION_BLOCK "Jdrk_RS_WS_N01_8"   // FB31, SCL
{ S7_Optimized_Access := 'TRUE' }
VERSION : 0.1
   VAR_OUTPUT
      Temperature : Real;
   END_VAR
   VAR_IN_OUT
      mb_query : "mb_query";
   END_VAR
   VAR
      sb : "mb_station_block_udt";
   END_VAR
   VAR RETAIN
      offset : Real;
   END_VAR
   VAR_TEMP
      tmp : Int;
   END_VAR
BEGIN
   // JDRK - RS-WS-N01-8 - Temperature and Humidity sensor

   "mb_station_block_header"(sb := #sb, mb_query := #mb_query);

   #mb_query(mb_addr := 1,
             mode := #mb_query.c.read.input_reg,
             data_addr := 1,
             data_ptr := #tmp);

   IF #mb_query.Done THEN
       #Temperature := INT_TO_REAL(#tmp) / 10 + #offset;
   END_IF;

   "mb_station_block_footer"(sb := #sb, mb_query := #mb_query);
END_FUNCTION_BLOCK

// folder: Library/Modbus/Station blocks/sb Untested/K

FUNCTION_BLOCK "keller_pressure_transmitters"   // FB99, SCL
{ S7_Optimized_Access := 'TRUE' }
VERSION : 0.1
   VAR_INPUT
      mb_addr : USInt;
   END_VAR
   VAR_IN_OUT
      mb_query : "mb_query";
   END_VAR
   VAR
      sb : "mb_station_block_udt";
      data : Struct
         pressure_sensor_1 : Real;
         pressure_sensor_2 : Real;
         temperature : Real;
         temperature_sensor_1 : Real;
         temperature_sensor_2 : Real;
      END_STRUCT;
   END_VAR
BEGIN
   // Keller, Series 30 and Series 40 - Pressure transmitters
   // 
   // http://www.keller-druck.com/picts/pdf/engl/comm_protocol_e.pdf

   "mb_station_block_header"(sb := #sb, mb_query := #mb_query);

   #mb_query(mb_addr := #mb_addr,
             mode := #mb_query.c.read.holding_reg,
             data_addr := 2,
             data_ptr := #data);

   "mb_station_block_footer"(sb := #sb, mb_query := #mb_query);
END_FUNCTION_BLOCK

// folder: Library/Modbus/Station blocks/sb Untested/K/Krohne

FUNCTION_BLOCK "Krohne_Optisonic"   // FB34, SCL
{ S7_Optimized_Access := 'TRUE' }
VERSION : 0.1
   VAR_INPUT
      mb_addr : UInt;
   END_VAR
   VAR_IN_OUT
      mb_query : "mb_query";
   END_VAR
   VAR
      sb : "mb_station_block_udt";
      data : Struct
         "Temperature process value" : Real;
         "Dynamic Viscosity at Process conditions" : Real;
         "Density Process" : Real;
         "Flow Process" : Real;
         "Velocity Process" : Real;
         "Speed of Sound" : Real;
      END_STRUCT;
   END_VAR
BEGIN
   // Krohne - Optisonic V6
   // 

   "mb_station_block_header"(sb := #sb,
                             mb_query := #mb_query);
   #mb_query.mb_addr := #mb_addr;

   #mb_query.mode := #mb_query.c.read.holding_reg;
   #mb_query(data_addr := 7050,
             data_ptr := #data);

   "mb_station_block_footer"(sb := #sb,
                             mb_query := #mb_query);
END_FUNCTION_BLOCK

FUNCTION_BLOCK "Krohne_MFC_300"   // FB100, SCL
TITLE = Krohne MFC 300
{ S7_Optimized_Access := 'TRUE' }
AUTHOR : OlaBjornli
FAMILY : modbus
VERSION : 0.1
// Coriolise flow meter
   VAR_INPUT
      mb_addr : UInt;
   END_VAR
   VAR_OUTPUT
      Temperature : Real;   // [degree C]
   END_VAR
   VAR_IN_OUT
      mb_query : "mb_query";
   END_VAR
   VAR
      sb : "mb_station_block_udt";
      read1 : Struct
         "Flow Velocity" : Real;   // [m/s]
         "Volume Flow" : Real;   // [m3/s]
         "Mass Flow" : Real;   // [kg/s]
         Temperature : Real := 273.15;   // [K]
         Density : Real;   // [kg/m3]
         Concentration_1 : Real;
         Concentration_2_or_Diagnosis_3 : Real;
         Concentration_Flow_1 : Real;
         Concentration_Flow_2 : Real;
         Diagnosis_1 : Real;
         Diagnosis_2 : Real;
         Display_Channel_1 : Real;
         Display_Channel_2 : Real;
         Operating_time : Real;   // [s]
      END_STRUCT;
      write1_settings : Struct
         Counter_1_Function : UInt;
         Counter_1_Measurement : UInt;
         Counter_2_Function : UInt;
         Counter_2_Measurement : UInt;
         Counter_3_Function : UInt;
         Counter_3_Measurement : UInt;
      END_STRUCT;
      exec_write : Bool;
   END_VAR
BEGIN
   // Krohne - MFC 300 
   // Flowmeter
   // 
   // Web: http://cdn.krohne.com/dlc/AD_MFC300_Modbus_en_091124_4000744801_R01.pdf
   //
   // #settings :
   //    Counter Function:
   //       1 = Sum Counter
   //       2 = + Counter
   //       3 = - Counter
   //       0 = Off
   //    Counter Measurement:
   //       21 = Volume Flow [m3]
   //       22 = Mass Flow [kg]
   //       27 = Concentration Flow 1
   //       28 = Concentration Flow 2

   "mb_station_block_header"(sb := #sb, mb_query := #mb_query);
   #mb_query.mb_addr := #mb_addr;

   #mb_query(mode := #mb_query.c.mode.read,
             data_addr := 30001, // 30000 + 1 (error in datasheet)
             data_ptr := #read1);
   #Temperature := #read1.Temperature - 273.15;

   // The write query isn't executing continuously in case that will damage eeprom
   IF #exec_write THEN
       #mb_query(mode := #mb_query.c.mode.write,
                 data_addr := 40001, // 40000 + 1,
                 data_ptr := #write1_settings);
       #exec_write := NOT #mb_query.Done;
   END_IF;

   "mb_station_block_footer"(sb := #sb, mb_query := #mb_query);
END_FUNCTION_BLOCK

// folder: Library/Modbus/Station blocks/sb Untested/M

FUNCTION_BLOCK "Moxa_ioLogik_R1200"   // FB36, SCL
{ S7_Optimized_Access := 'TRUE' }
VERSION : 0.1
   VAR_INPUT
      mb_addr : UInt;
   END_VAR
   VAR_IN_OUT
      mb_query : "mb_query";
   END_VAR
   VAR
      sb : "mb_station_block_udt";
      in : Array[0..15] of Bool;
      out : Array[0..15] of Bool;
   END_VAR
BEGIN
   // Moxa - ioLogik R1200
   // 
   // https://www.moxa.com/doc/man/ioLogik_R1200_Series_UM_e3.1.pdf

   "mb_station_block_header"(sb := #sb, mb_query := #mb_query);
   #mb_query.mb_addr := #mb_addr;

   #mb_query(mode := #mb_query.c.read.discrete_input,
             data_addr := 0,
             data_ptr := #in);

   #mb_query(mode := #mb_query.c.write.discrete_output,
             data_addr := 16#140,
             data_ptr := #out);

   "mb_station_block_footer"(sb := #sb, mb_query := #mb_query);
END_FUNCTION_BLOCK

FUNCTION_BLOCK "MTS_sensors_M_Series"   // FB37, SCL
{ S7_Optimized_Access := 'TRUE' }
VERSION : 0.1
   VAR_INPUT
      mb_addr : UInt;
   END_VAR
   VAR_OUTPUT
      level : Real;
      temperature : Real;
   END_VAR
   VAR_IN_OUT
      mb_query : "mb_query";
   END_VAR
   VAR
      sb : "mb_station_block_udt";
      read : Struct
         product_level : DInt;
         Interface_level : DInt;
         roof_level : DInt;
         temperature : Array[1..5] of DInt;
         temperature_avg : DInt;
      END_STRUCT;
   END_VAR
BEGIN
   // MTS sensors - M-Series - Liquid-Level Sensors
   // Web: http://www.mtssensors.com/fileadmin/media/pdfs/550791.pdf

   "mb_station_block_header"(sb := #sb, mb_query := #mb_query);
   #mb_query.mb_addr := #mb_addr;

   #mb_query.mode := #mb_query.c.mode.read;
   #mb_query(data_addr := 30001, data_ptr := #read);

   "mb_station_block_footer"(sb := #sb, mb_query := #mb_query);

   #level := DINT_TO_REAL(#read.product_level) * 0.001;
   #temperature := DINT_TO_REAL(#read.temperature_avg) * 0.0001;
END_FUNCTION_BLOCK

FUNCTION_BLOCK "masibus_85XX"   // FB86, SCL
{ S7_Optimized_Access := 'TRUE' }
VERSION : 0.1
   VAR_INPUT
      mb_addr : USInt;
   END_VAR
   VAR_IN_OUT
      mb_query : "mb_query";
   END_VAR
   VAR
      sb : "mb_station_block_udt";
      read1 : Struct
         channel : Array[1..24] of Int;
         Ambient_PV : Int;
         digital_output_status : DWord;
         alarm : Array[1..2] of DWord;
         control_status : DWord;
         alarm_blink_status : Array[1..2] of DWord;
         alarm_LED_status : Array[1..2] of DWord;
      END_STRUCT;
      write1_labels : Array[1..24] of String[6];
      write2_input_type : Array[1..24] of USInt;
   END_VAR
BEGIN
   // Masibus - 85XX+
   // SCANNER / DAQ
   // REF NO: m83B/om/101
   // http://www.masibus.com/Pmanual/Data_Acquisition/
   // Enhanced_Multi-Channel_Scanners/85XX+_User_Manual

   "mb_station_block_header"(sb := #sb, mb_query := #mb_query);
   #mb_query.mb_addr := #mb_addr; // Device address.

   #mb_query.mode := #mb_query.c.mode.read;
   #mb_query(data_addr := 30001, data_ptr := #read1);

   #mb_query.mode := #mb_query.c.mode.write;
   #mb_query(data_addr := 42204, data_ptr := #write1_labels);
   #mb_query(data_addr := 40097, data_ptr := #write2_input_type);

   "mb_station_block_footer"(sb := #sb, mb_query := #mb_query);

   (*

   #  : Type
   ------------
   00 : None
   01 : E-tc
   02 : J-tc
   03 : K-tc
   04 : T-tc
   05 : B-tc
   06 : R-tc 
   07 : S-tc
   08 : n-tc
   09 : RDT
   10 : Cu53
   11 : Ni120
   12 : -10.20mV
   13 : 0-100mV
   14 : 4-20mA
   15 : 0-20mA
   16 : 0-5V
   17 : 1-5V
   18 : 0-10V
   19 : Dig.inp

   *)
END_FUNCTION_BLOCK

// folder: Library/Modbus/Station blocks/sb Untested/M/Mettler

FUNCTION_BLOCK "mettler_toledo_IND560_loadTargetValue"   // FB87, SCL
{ S7_Optimized_Access := 'TRUE' }
VERSION : 0.1
   VAR_INPUT
      iValue : Real;
   END_VAR
   VAR_OUTPUT
      qDone : Bool;
   END_VAR
   VAR_IN_OUT
      "M" : "mettlerToledoInd560Udt";
      sb : "mb_station_block_udt";
   END_VAR
   VAR
      state : Int;
      old_value : Real;
      slot : USInt;
   END_VAR
   VAR CONSTANT
      NONE_AVAILABLE : USInt := 0;
   END_VAR
BEGIN
   // Load target value, for scale 1. Page 143, table B-6

   CASE #state OF

       0:  // Waiting for start.
           #qDone := false;
           #state +=
           BOOL_TO_INT(#old_value <> #iValue);

       1:  // Wait for available msg. slot
           #slot := "reqMsgSlot"(#"M".occupiedMsgSlots);
           #state += BOOL_TO_INT(#slot <> #NONE_AVAILABLE);

       2:  // #1 PLC loads floating point value first
           #"M".writeMsgSlot[#slot].cmd := 0;
           #"M".writeMsgSlot[#slot].data := #iValue;
           #state += 1;
       3:
           #state += BOOL_TO_INT(#"M".queryDone.write);

       4:  // #2 PLC sends command to set target 1 cutoff value 
           #"M".writeMsgSlot[#slot].cmd := 110;
           #state += 1;
       5:
           #state += BOOL_TO_INT(#"M".queryDone.write);

       6:  // #3 IND560 terminal sees new command, loads the value into the target
           //    and ends a return message to indicate the new target value.
           #state +=
           BOOL_TO_INT(#"M".queryDone.read
                       AND #"M".run.cmdAck[#slot] = 1
                       AND #"M".run.PF[#slot] = 13
                       AND #"M".readMsgSlot[#slot].data = #"M".writeMsgSlot[#slot].data);

       7:  // #4  PLC instructs IND560 terminal to start â€œusingâ€ new target value
           #"M".writeMsgSlot[#slot].cmd := 114;
           #state += 1;
       8:
           #state += BOOL_TO_INT(#"M".queryDone.write);

       9:  // #5 IND560 terminal sees new command
           #"M".writeMsgSlot[#slot].cmd := 0;

           #state +=
           BOOL_TO_INT(#"M".queryDone.read
                       AND #"M".run.cmdAck[#slot] = 2
                       AND #"M".run.PF[#slot] = 30
                       AND #"M".readMsgSlot[#slot].data = 0);

       ELSE: // Back to start.
           #"M".occupiedMsgSlots[#slot] := false; // Release msg. slot.
           #state := 0;
           #qDone := true;
           // The start signal should need to be set back false before next
           // exec. else the sequence will start over.
   END_CASE;
   #old_value := #iValue;

   // 
   IF #sb.out.Communication_error THEN
       #state := 0;
       IF #slot <> #NONE_AVAILABLE THEN
           #"M".writeMsgSlot[#slot].cmd := 0;
           "releaseMsgSlot"(slot := #slot,
                            mem := #"M".occupiedMsgSlots);
       END_IF;
   END_IF;
END_FUNCTION_BLOCK

FUNCTION_BLOCK "mettler_toledo_IND560"   // FB88, SCL
{ S7_Optimized_Access := 'TRUE' }
VERSION : 0.1
   VAR_IN_OUT
      mb_query : "mb_query";
   END_VAR
   VAR
      mb_addr : UInt := 255;
      sb : "mb_station_block_udt";
      "M" : "mettlerToledoInd560Udt";   // Shared data
      loadTargetValue : "mettler_toledo_IND560_loadTargetValue";
      s : USInt;
   END_VAR
   VAR_TEMP
      c : Int;
   END_VAR
BEGIN
   // Mettler Toledo IND560 - Weighing Terminal

   // WARNING: This SB is just a draft and the block probably include errors !!

   // Necessary settings: ()
   // PLC -> Eth/IP - Modbus TCP -> IP-address
   // PLC -> Eth/IP - Modbus TCP -> Subnet-mask
   // PLC -> Data Format -> Byte order : standard
   // PLC -> Data Format -> Format     : Floating Point 

   // - Modbus tcp:
   //   https://bradysystems.com/wp-content/uploads/2012/10/IND560-PLC-Interface-Manual.pdf
   // - Product overview:
   //   http://www.atsackfillers.mobi/assets/ind560_ug_en_71209396_r04.pdf

   REGION Modbus
       "mb_station_block_header"(sb := #sb,
                                 mb_query := #mb_query);
       #mb_query.mb_addr := #mb_addr;

       #mb_query(mode := #mb_query.c.mode.read,
                 data_addr := 400001,
                 data_ptr := #"M".readMsgSlot,
                 Done => #"M".queryDone.read);

       #mb_query(mode := #mb_query.c.mode.write,
                 data_addr := 401026,
                 data_ptr := #"M".writeMsgSlot,
                 Done => #"M".queryDone.write);

       "mb_station_block_footer"(sb := #sb,
                                 mb_query := #mb_query);
   END_REGION

   REGION Read data-fix     
       // Extract bits in word in to a numbers.
       FOR #c := 1 TO 4 DO
           #"M".run.PF[#c].%X0 := #"M".readMsgSlot[#c].cmdRespons.FP_1;
           #"M".run.PF[#c].%X1 := #"M".readMsgSlot[#c].cmdRespons.FP_2;
           #"M".run.PF[#c].%X2 := #"M".readMsgSlot[#c].cmdRespons.FP_3;
           #"M".run.PF[#c].%X3 := #"M".readMsgSlot[#c].cmdRespons.FP_4;
           #"M".run.PF[#c].%X4 := #"M".readMsgSlot[#c].cmdRespons.FP_5;

           #"M".run.cmdAck[#c].%X0 := #"M".readMsgSlot[#c].cmdRespons.cmdAck1;
           #"M".run.cmdAck[#c].%X1 := #"M".readMsgSlot[#c].cmdRespons.cmdAck2;
       END_FOR;
   END_REGION


   #loadTargetValue(M := #"M",
                    sb := #sb);




   #"M".queryDone.write := false;
   #"M".queryDone.read := false;
END_FUNCTION_BLOCK

FUNCTION "releaseMsgSlot" : Void   // FC17, SCL
{ S7_Optimized_Access := 'TRUE' }
VERSION : 0.1
   VAR_IN_OUT
      slot : USInt;
      mem : Array[*] of Bool;
   END_VAR
   VAR_TEMP
      c : Int;
   END_VAR
BEGIN

   IF #slot <> 0 THEN
       #mem[#slot] := false;
   END_IF;
END_FUNCTION

FUNCTION "reqMsgSlot" : USInt   // FC18, SCL
{ S7_Optimized_Access := 'TRUE' }
VERSION : 0.1
   VAR_IN_OUT
      mem : Array[*] of Bool;
   END_VAR
   VAR_TEMP
      c : Int;
   END_VAR
BEGIN
   // Find first entry inside mem that is false.
   // set the entry to true and return the index. 

   #reqMsgSlot := 0;
   FOR #c := LOWER_BOUND(ARR := #mem, DIM := 1) TO
       UPPER_BOUND(ARR := #mem, DIM := 1)
   DO
       IF NOT #mem[#c] THEN
           #mem[#c] := true;
           #reqMsgSlot := INT_TO_USINT(#c);
           RETURN;
       END_IF;
   END_FOR;
END_FUNCTION

// folder: Library/Modbus/Station blocks/sb Untested/N

FUNCTION_BLOCK "Novus_tht"   // FB38, SCL
{ S7_Optimized_Access := 'TRUE' }
VERSION : 0.1
   VAR_INPUT
      mb_addr : USInt;
   END_VAR
   VAR_OUTPUT
      temperature : Int;
      humidity : Int;
   END_VAR
   VAR_IN_OUT
      mb_query : "mb_query";
   END_VAR
   VAR
      sb : "mb_station_block_udt";
      serial_number : DWord;
      raw_values : Struct
         temp : Int;
         hum : Int;
      END_STRUCT;
   END_VAR
BEGIN
   // - Novus - RHT (Temperature transmitter)
   // - http://www.novusautomation.com/downloads/Arquivos/v10x_b_manual_rht_wm-dm-p10_485_lcd_%20english.pdf

   "mb_station_block_header"(sb := #sb, mb_query := #mb_query);
   #mb_query.mb_addr := #mb_addr;

   #mb_query.mode := #mb_query.c.read.holding_reg;
   #mb_query(data_addr := 7, data_ptr := #raw_values);
   #mb_query(data_addr := 0, data_ptr := #serial_number);

   "mb_station_block_footer"(sb := #sb, mb_query := #mb_query);

   #temperature := #raw_values.temp / 10;
   #humidity := #raw_values.hum / 10;
END_FUNCTION_BLOCK

// folder: Library/Modbus/Station blocks/sb Untested/O

FUNCTION_BLOCK "Onicon_F5100"   // FB39, SCL
{ S7_Optimized_Access := 'TRUE' }
VERSION : 0.1
   VAR_INPUT
      mb_addr : USInt;
   END_VAR
   VAR_IN_OUT
      mb_query : "mb_query";
   END_VAR
   VAR
      sb : "mb_station_block_udt";
      reset : Bool;
      query1 : Struct
         flow_total : UDInt;
      END_STRUCT;
      query2 : Struct
         flow_rate : Real;
         temperature : Real;
      END_STRUCT;
   END_VAR
BEGIN
   // Onicon - F-5100
   // http://www.onicon.com/pdfs/0669-7-F-5100-MOD-Network-Interface-Installation-Guide-09-15.pdf

   "mb_station_block_header"(sb := #sb, mb_query := #mb_query);
   #mb_query.mb_addr := #mb_addr;

   #mb_query.data_addr := 312; // 313 - 1
   IF #reset THEN
       #query1.flow_total := 0;
       #mb_query(mode := #mb_query.c.write.holding_reg,
                 data_ptr := #query1.flow_total);
       IF #mb_query.stat.done THEN
           #reset := false;
       END_IF;
   ELSE
       #mb_query(mode := #mb_query.c.read.holding_reg, data_ptr := #query1);
   END_IF;

   #mb_query(mode := #mb_query.c.read.holding_reg,
             data_addr := 578, // 579 - 1,
             data_ptr := #query2);

   "mb_station_block_footer"(sb := #sb, mb_query := #mb_query);
END_FUNCTION_BLOCK

// folder: Library/Modbus/Station blocks/sb Untested/P

FUNCTION_BLOCK "Phoenix_Contact_UPS"   // FB40, SCL
{ S7_Optimized_Access := 'TRUE' }
VERSION : 0.1
   VAR_INPUT
      mb_addr : UInt;
   END_VAR
   VAR_IN_OUT
      mb_query : "mb_query";
   END_VAR
   VAR
      sb : "mb_station_block_udt";
      read1 : Struct
         remote : Word;
         BatteryMode : Word;
         ShutdownEvent : Word;
         BatteryCharging : Word;
      END_STRUCT;
      read2 : Struct
         OutputVoltage_mV : UInt;
      END_STRUCT;
      read3 : Struct
         SocStateOfCharge : UInt;   // [%]
         SocResidualBackupTimeM : UInt;   // Minute
      END_STRUCT;
      read4 : Struct
         BatteryVoltage_mV : UInt;
         BatteryTemperature : UInt;   // Kelvin
         OutputVoltage2_mV : UInt;
         SocResidualBackupTimeS : UInt;
         BatteryNomCapacityWs : UInt;
      END_STRUCT;
      read5 : Struct
         BatteryDischaCurrent : UInt;
         BatteryDetectedUnits : UInt;
         BatteryNomCapacitymAh : UInt;
         BatteryInstalledType : UInt;
      END_STRUCT;
      read6_Alarm : Struct
         x08 : Bool;
         x09_no_battery : Bool;
         x10_inconsistent_technology : Bool;
         x11_overload_cutoff : Bool;
         "x12_Low_battery_(Voltage)" : Bool;
         "x13_Low_battery_(Charge)" : Bool;
         "x14_Low_battery_(Time)" : Bool;
         x15 : Bool;
         "x00_End_of_life_(SOH)" : Bool;
         x01 : Bool;
         x02 : Bool;
         x03 : Bool;
         "x04_End_of_life_(Resitance)" : Bool;
         "x05_Endof_life_(Resitance)" : Bool;
         "x06_End_of_life_(Time)" : Bool;
         "x07_End_of_life_(Voltage)" : Bool;
      END_STRUCT;
   END_VAR
BEGIN
   // Phoenix Contact - UPS
   // QUINT UPS-IQ, TRIO-UPS
   // Web: https://media.digikey.com/pdf/Data%20Sheets/
   //      Phoenix%20Contact%20PDFs/2320461_Ds.pdf

   "mb_station_block_header"(sb := #sb, mb_query := #mb_query);
   #mb_query.mb_addr := #mb_addr;

   #mb_query.mode := #mb_query.c.read.holding_reg;
   #mb_query(data_addr := 29696, data_ptr := #read1);
   #mb_query(data_addr := 29745, data_ptr := #read2);
   #mb_query(data_addr := 29749, data_ptr := #read3);
   #mb_query(data_addr := 29792, data_ptr := #read4);
   #mb_query(data_addr := 29798, data_ptr := #read5);
   #mb_query(data_addr := 29840, data_ptr := #read6_Alarm);

   "mb_station_block_footer"(sb := #sb, mb_query := #mb_query);
END_FUNCTION_BLOCK

// folder: Library/Modbus/Station blocks/sb Untested/P/ProMinent

FUNCTION_BLOCK "ProMinent_Dulcometer"   // FB125, SCL
{ S7_Optimized_Access := 'TRUE' }
VERSION : 0.1
   VAR_INPUT
      mb_addr : USInt;
   END_VAR
   VAR_IN_OUT
      mb_query : "mb_query";
   END_VAR
   VAR
      sb : "mb_station_block_udt";
      read1 : Array[1..2] of Struct
         actual_measured_value : Real;
         Controller_Actuating_value : Int;
         Temperature : Int;
         "Actual Set Point" : Real;
         Actual_ExternalDisturbanceValue : UInt;
         Status : Word;
         Warnings : Word;
      END_STRUCT;
      write1 : Struct
         "a" : Bool;
      END_STRUCT;
      serial_number : UDInt;
   END_VAR
BEGIN
   // ProMient - DULCOMETER
   // Multi-parameter Controller diaLog DACa

   "mb_station_block_header"(sb := #sb, mb_query := #mb_query);
   #mb_query.mode := #mb_addr;

   #mb_query.mode := #mb_query.c.read.holding_reg;
   #mb_query(data_addr := 16#63, data_ptr := #read1[1]);
   #mb_query(data_addr := 16#70, data_ptr := #read1[2]);
   #mb_query(data_addr := 16#91, data_ptr := #serial_number);

   "mb_station_block_footer"(sb := #sb, mb_query := #mb_query);

   (* Default settings:
   parity: Odd  
   stop bits: 1 
   Baud rate: 19200 
   *)
END_FUNCTION_BLOCK

// folder: Library/Modbus/Station blocks/sb Untested/P/Produal

FUNCTION_BLOCK "produal_KLH_M"   // FB42, SCL
{ S7_Optimized_Access := 'TRUE' }
VERSION : 0.1
   VAR_INPUT
      mb_addr : USInt;
   END_VAR
   VAR_OUTPUT
      temperature : Real;
      humidity : Real;
      potentiometer : Real;
   END_VAR
   VAR_IN_OUT
      mb_query : "mb_query";
   END_VAR
   VAR
      sb : "mb_station_block_udt";
      write1_calibration : Struct
         temp_offset : Int;
         humidity_offset : Int;
      END_STRUCT;
      read1 : Struct
         temperature : Int;
         humidity : UInt;
         y : Array[1..4] of UInt;
         potentiometer : Int;   // %
      END_STRUCT;
   END_VAR
BEGIN
   // Produal - KLH-M
   // Product number: 1132600
   // http://www.produal.com/shop/web_humidity_transmitters/sku-1132600

   "mb_station_block_header"(sb := #sb, mb_query := #mb_query);
   #mb_query.mb_addr := #mb_addr;

   #mb_query(mode := #mb_query.c.mode.read,
             data_addr := 30001,
             data_ptr := #read1);

   #mb_query(mode := #mb_query.c.mode.write,
             data_addr := 40006,
             data_ptr := #write1_calibration); // temp. and humidity  

   "mb_station_block_footer"(sb := #sb, mb_query := #mb_query);

   #temperature := INT_TO_REAL(#read1.temperature) * 0.1;
   #humidity := UINT_TO_REAL(#read1.humidity); // 0-100%
   #potentiometer := INT_TO_REAL(#read1.potentiometer) * 0.1;
END_FUNCTION_BLOCK

FUNCTION_BLOCK "produal_TEHR_M"   // FB43, SCL
{ S7_Optimized_Access := 'TRUE' }
VERSION : 0.1
   VAR_INPUT
      mb_addr : USInt;
      calibration_offset : Int;   // mbar
   END_VAR
   VAR_OUTPUT
      temperature : Real;   // Â°C
      analogue_output : Real;   // V
      potentiometer : Real;   // %
   END_VAR
   VAR_IN_OUT
      mb_query : "mb_query";
   END_VAR
   VAR
      sb : "mb_station_block_udt";
      r1 : Struct
         temperature : Int;
         analogue_output : UInt;
         potentiometer : Int;
      END_STRUCT;
   END_VAR
BEGIN
   // Produal - TEHR-M - Temperatur transmitter.
   // Product: 117Z190 - Pt1000 EN 60751/B
   // http://www.produal.com/shop/web_bus_temperature_transmitters/
   // sku-117Z190?hiddenAttributes_sensor_output=sensor_output_modbus&saf=true

   "mb_station_block_header"(sb := #sb,
                             mb_query := #mb_query);
   #mb_query.mb_addr := #mb_addr;

   #mb_query(mode := #mb_query.c.mode.read,
             data_addr := 30001,
             data_ptr := #r1);

   #mb_query(mode := #mb_query.c.mode.write,
             data_addr := 40001,
             data_ptr := #calibration_offset);

   "mb_station_block_footer"(sb := #sb,
                             mb_query := #mb_query);

   #temperature := INT_TO_REAL(#r1.temperature) * 0.1;
   #analogue_output := UINT_TO_REAL(#r1.analogue_output);
   #potentiometer := INT_TO_REAL(#r1.potentiometer) * 0.1;
END_FUNCTION_BLOCK

// folder: Library/Modbus/Station blocks/sb Untested/R

FUNCTION_BLOCK "Rotork_Mk_3_option_card"   // FB44, SCL
{ S7_Optimized_Access := 'TRUE' }
VERSION : 0.1
   VAR_INPUT
      mb_addr : UInt;
   END_VAR
   VAR_IN_OUT
      mb_query : "mb_query";
   END_VAR
   VAR
      sb : "mb_station_block_udt";
      read1 : Struct
         x00_actuator_moving : Bool;
         "x01_Close position limit" : Bool;
         "x02_Open position limit" : Bool;
         "x03_Valve running close" : Bool;
         "x04_Valve running open" : Bool;
         "x05_Selector in remote" : Bool;
         "x06_Selector in local stop" : Bool;
         "x07_Selector in local" : Bool;
         "x08_Thermostat tripped" : Bool;
         "x09_Monitor relay" : Bool;
         "x10_Valve obstructed" : Bool;
         "x11_Valve jammed" : Bool;
         "x12_Manual movement" : Bool;
         "x13_MIT_Interrupter timer" : Bool;
         "x14_Position control enabled" : Bool;
         "x15_Watchdog Recovery" : Bool;
         "x16_Battery low" : Bool;
         "x17_Open Interlock input active" : Bool;
         "x18_Close Interlock input active" : Bool;
         "x19_Hard wired input DI-1 (open)" : Bool;
         "x20_Hard wired input DI-2 (close)" : Bool;
         "x21_Hard wired input DI-3 (stop)" : Bool;
         "x22_Hard wired input DI-4 (ESD)" : Bool;
         x23 : Bool;
         x24 : Bool;
         x25 : Bool;
         "x26_Control contention" : Bool;
         "x27_Partial stroke test in progress" : Bool;
         "x28_Partial stroke test error" : Bool;
         "x29_General alarm" : Bool;
         x30 : Bool;
         x31 : Bool;
      END_STRUCT;
      read2 : Struct
         instantaneous_torque : Int;
         valve_position : Int;   // x10 %
         analogue_input : Int;
      END_STRUCT;
      write1 : Struct
         stop : Bool;
         close : Bool;
         open : Bool;
         emergency_shut_down : Bool;
         output_DO_1 : Bool;
         output_DO_2 : Bool;
         output_DO_3 : Bool;
         output_DO_4 : Bool;
      END_STRUCT;
      write2 : Struct
         actuator_digital_control : Bool;
         position_demand_output : Bool;
      END_STRUCT;
      actuator_tag_name : String[12];
      action_on_loss_of_comms : Int;
   END_VAR
BEGIN
   // Rotork  - Mk 3 Option Card

   // http://www.rotork.com/en/product/index/modbusliterature
   // Publication PUB091-004-00_0715

   "mb_station_block_header"(sb := #sb, mb_query := #mb_query);
   #mb_query.mb_addr := #mb_addr;

   #mb_query.mode := #mb_query.c.read.discrete_input;
   #mb_query(data_addr := 0, data_ptr := #read1);

   #mb_query.mode := #mb_query.c.read.holding_reg;
   #mb_query(data_addr := 2, data_ptr := #read2);
   #mb_query(data_addr := 26, data_ptr := #actuator_tag_name);

   #mb_query.mode := #mb_query.c.write.discrete_output;
   #mb_query(data_addr := 0, data_ptr := #write1);

   #mb_query.mode := #mb_query.c.write.holding_reg;
   // 0=No-Action, 1=Open, 3=Close, 5=Stop, 7=Position
   #mb_query(data_addr := 7, data_ptr := #action_on_loss_of_comms);
   #mb_query(data_addr := 5, data_ptr := #write2);

   "mb_station_block_footer"(sb := #sb, mb_query := #mb_query);
END_FUNCTION_BLOCK

// folder: Library/Modbus/Station blocks/sb Untested/S

FUNCTION_BLOCK "SensorsONE_DCT_531"   // FB52, SCL
{ S7_Optimized_Access := 'TRUE' }
VERSION : 0.1
   VAR_INPUT
      mb_addr : UInt;
   END_VAR
   VAR_IN_OUT
      mb_query : "mb_query";
   END_VAR
   VAR
      sb : "mb_station_block_udt";
      data : Struct
         serial_number : UDInt;
         date_last_calibration : UDInt;
         upper_range_pressure : Real;
         lower_range_pressure : Real;
         actual_pressure : Real;
         max_pressure : Real;
         min_pressure : Real;
         upper_range_temperature : Real;
         lower_range_temperature : Real;
         actual_temperature : Real;
         max_temperature : Real;
         min_temperature : Real;
      END_STRUCT;
   END_VAR
BEGIN
   // SensorsONE - DCT 531
   // 
   // https://www.sensorsone.com/dct-531-modbus-rtu-rs485-pressure-sensor/

   "mb_station_block_header"(sb := #sb, mb_query := #mb_query);
   #mb_query.mb_addr := #mb_addr;

   #mb_query.mode := #mb_query.c.read.input_reg;
   #mb_query(data_addr := 0, data_ptr := #data);

   "mb_station_block_footer"(sb := #sb, mb_query := #mb_query);
END_FUNCTION_BLOCK

FUNCTION_BLOCK "Sierra_thermal_mass_flow_meters"   // FB61, SCL
{ S7_Optimized_Access := 'TRUE' }
VERSION : 0.1
   VAR_INPUT
      mb_addr : UInt;
      reset_totalizer : Bool := 1;
   END_VAR
   VAR_IN_OUT
      mb_query : "mb_query";
   END_VAR
   VAR
      sb : "mb_station_block_udt";
      data : Struct
         flow : Real;
         totalizer : DInt;
      END_STRUCT;
      serial_number : String[12];
   END_VAR
   VAR_TEMP
      "int" : Int;
   END_VAR
BEGIN
   // Sierra - 600/700 Series - Thermal mass flow meters
   // Models: 620S, 620S-BT, 640S, 760S, 780S, and 780S-UHP

   // Web: https://www.ccontrols.com/support/dp/600-700-modbus-instruction-manual.pdf

   "mb_station_block_header"(sb := #sb, mb_query := #mb_query);
   #mb_query.mb_addr := #mb_addr;

   #mb_query.mode := #mb_query.c.mode.read;
   #mb_query(data_addr := 40001, data_ptr := #data);
   #mb_query(data_addr := 40016, data_ptr := #serial_number);

   IF #reset_totalizer THEN
       #mb_query.mode := #mb_query.c.mode.write;
       #"int" := 1;
       #mb_query(data_addr := 40008, data_ptr := #"int");
   END_IF;

   "mb_station_block_footer"(sb := #sb, mb_query := #mb_query);
END_FUNCTION_BLOCK

FUNCTION_BLOCK "Smart_biene_sb_hl"   // FB62, SCL
{ S7_Optimized_Access := 'TRUE' }
VERSION : 0.1
   VAR_INPUT
      mb_addr : UInt;
   END_VAR
   VAR_IN_OUT
      mb_query : "mb_query";
   END_VAR
   VAR
      s : "mb_station_block_udt";
      data : Struct
         "Min measuring range" : Word;
         "Max measuring range" : Word;
         "Pressure Value" : Word;
         "High Pressure" : Word;
         "Low Pressure" : Word;
         stat : Word;
         model : String[12];
         serial : String[12];
         unit : Int;
      END_STRUCT;
      "a" : Struct
         x08 : Bool;
         x09 : Bool;
         x10 : Bool;
         x11 : Bool;
         x12 : Bool;
         x13 : Bool;
         x14 : Bool;
         x15 : Bool;
         x00 : Bool;
         x01 : Bool;
         x02 : Bool;
         x03 : Bool;
         x04 : Bool;
         x05 : Bool;
         x06 : Bool;
         x07 : Bool;
      END_STRUCT;
   END_VAR
BEGIN
   // Smart Biene - SB-HL - Hydrostatic Level Transmitter
   // 
   // http://smartbiene.com/images/pdf/hydrostatic-level/Hydrostatic%20level-SP-HL-01-ModbusRTU.pdf

   "mb_station_block_header"(sb := #s, mb_query := #mb_query);
   #mb_query.mb_addr := #mb_addr;

   #mb_query.mode := #mb_query.c.read.holding_reg;
   #mb_query(data_addr := 0, data_ptr := #data);

   "mb_station_block_footer"(sb := #s, mb_query := #mb_query);

   (*
   Unit:
   0-mbar
   1-bar
   2-PSI
   3-KPa
   4-MPa
   5-Kg/cm2
   6-mmHg
   7-mmH2O
   8-inHg
   9-inH2O 
   *)
END_FUNCTION_BLOCK

FUNCTION_BLOCK "Socomec_diris"   // FB63, SCL
{ S7_Optimized_Access := 'TRUE' }
VERSION : 0.1
   VAR_INPUT
      mb_addr : USInt;
      old_mapping : Bool;
      zero_comm_err : Bool;
   END_VAR
   VAR_OUTPUT
      data : Struct
         voltage_L_L : Array[1..3] of Real;   // 1->L1-L2, 2->L2-L3, 3->L3-L1
         voltage_L_N : Array[1..3] of Real;
         frequency : Real;
         current : Array[1..3] of Real;
         neutral_current : Real;
         sum_active_power : Real;
         sum_reactive_power : Real;
         sum_apparent_power : Real;
         sum_power_factor : Real;   // -: leading and + : lagging
         power_active : Array[1..3] of Real;
         power_reactive : Array[1..3] of Real;
         power_apparent : Array[1..3] of Real;
         power_factor : Array[1..3] of Real;
      END_STRUCT;
   END_VAR
   VAR_IN_OUT
      mb_query : "mb_query";
   END_VAR
   VAR
      sb : "mb_station_block_udt";
      read2_temperature : DInt;
   END_VAR
   VAR_TEMP
      c : Int;
      read1 : Struct
         voltage_L_L : Array[1..3] of DInt;   // 1->L1-L2, 2->L2-L3, 3->L3-L1
         voltage_L_N : Array[1..3] of DInt;
         frequency : DInt;
         current : Array[1..3] of DInt;
         neutral_current : DInt;
         sum_active_power : DInt;
         sum_reactive_power : DInt;
         sum_apparent_power : DInt;
         sum_power_factor : DInt;   // -: leading and + : lagging
         power_active : Array[1..3] of DInt;
         power_reactive : Array[1..3] of DInt;
         power_apparent : Array[1..3] of DInt;
         power_factor : Array[1..3] of DInt;
      END_STRUCT;
   END_VAR
BEGIN
   // Socomec Diris A40/A41 - Power meter
   // https://www.socomec.com/files/live/sites/systemsite/files/SCP/
   // 6_gestion_energie/diris/diris_a40/536181B_GB_Ethernet.pdf

   // old_mapping:
   // http://www.ferrazshawmutsales.com/pdfs/cdr_27038_RS485_JBus-ModBus.pdf

   "mb_station_block_header"(sb := #sb, mb_query := #mb_query);
   #mb_query.mb_addr := #mb_addr;
   #mb_query.mode := #mb_query.c.read.holding_reg;

   #mb_query(data_addr := SEL(G := #old_mapping, IN0 := 50514, IN1 := 768),
             data_ptr := #read1);
   IF #mb_query.Done THEN
       FOR #c := 1 TO 3 DO
           #data.voltage_L_L[#c] := DINT_TO_REAL(#read1.voltage_L_L[#c]) / 100;
           #data.voltage_L_N[#c] := DINT_TO_REAL(#read1.voltage_L_N[#c]) / 100;
           #data.current[#c] := DINT_TO_REAL(#read1.current[#c]) / 1000;
           #data.power_active[#c] := DINT_TO_REAL(#read1.power_active[#c]) / 100;
           #data.power_reactive[#c] := DINT_TO_REAL(#read1.power_reactive[#c]) / 100;
           #data.power_apparent[#c] := DINT_TO_REAL(#read1.power_apparent[#c]) / 100;
           #data.power_factor[#c] := DINT_TO_REAL(#read1.power_factor[#c]) / 1000;
       END_FOR;
       #data.frequency := DINT_TO_REAL(#read1.frequency) / 100;
       #data.neutral_current := DINT_TO_REAL(#read1.neutral_current) / 100;
       #data.sum_active_power := DINT_TO_REAL(#read1.sum_active_power) / 100;
       #data.sum_reactive_power := DINT_TO_REAL(#read1.sum_reactive_power) / 100;
       #data.sum_apparent_power := DINT_TO_REAL(#read1.sum_apparent_power) / 100;
       #data.sum_power_factor := DINT_TO_REAL(#read1.sum_power_factor) / 1000;
   END_IF;

   IF NOT #old_mapping THEN
       #mb_query(data_addr := 51457, data_ptr := #read2_temperature);
   END_IF;

   "mb_station_block_footer"(sb := #sb, mb_query := #mb_query);

   IF #zero_comm_err AND #sb.out.Communication_error THEN
       FOR #c := 1 TO 3 DO
           #data.voltage_L_L[#c] := 0;
           #data.voltage_L_N[#c] := 0;
           #data.current[#c] := 0;
           #data.power_active[#c] := 0;
           #data.power_reactive[#c] := 0;
           #data.power_apparent[#c] := 0;
           #data.power_factor[#c] := 0;
       END_FOR;
       #data.frequency := 0;
       #data.neutral_current := 0;
       #data.sum_active_power := 0;
       #data.sum_reactive_power := 0;
       #data.sum_apparent_power := 0;
       #data.sum_power_factor := 0;

       #read2_temperature := 0;
   END_IF;
END_FUNCTION_BLOCK

FUNCTION_BLOCK "Sparling_Instruments_Tiger_Mag"   // FB64, SCL
{ S7_Optimized_Access := 'TRUE' }
VERSION : 0.1
   VAR_INPUT
      mb_addr : USInt;
   END_VAR
   VAR_IN_OUT
      mb_query : "mb_query";
   END_VAR
   VAR
      sb : "mb_station_block_udt";
      read1 : Struct
         flow : Real;   // 0.01 [Hz]
         total_fwd : UDInt;   // 0.1 [A]
         total_rev : UDInt;
         unit_flow : String[4];
         unit_total : String[4];
         total_registration : Real;
      END_STRUCT;
      serial_number : UDInt;
   END_VAR
BEGIN
   // Sparling Instruments - Tiger Mag 
   // FM656, FM657, FM626, FM627, FM626 Sanitary
   // http://www.sparlinginstruments.com/documents/IDS-TMEP-160323.PDF
   // Revision 160323

   "mb_station_block_header"(sb := #sb, mb_query := #mb_query);
   #mb_query.mb_addr := #mb_addr;

   #mb_query.mode := #mb_query.c.mode.read;
   #mb_query(data_addr := 30001, data_ptr := #read1);
   #mb_query(data_addr := 31003, data_ptr := #serial_number);

   "mb_station_block_footer"(sb := #sb, mb_query := #mb_query);

   (*
   Terminal RS-485 Bus:
   1-RX  -> A+
   2-TX  -> B-
   3-GND -> GND
   4-DTR -> N/A Not used

   Default comm. param:
   19200 bps, even parity. 
    Slave ID: 1.
   *)
END_FUNCTION_BLOCK

FUNCTION_BLOCK "Syxthsense_TEHR_M"   // FB70, SCL
TITLE = Syxthsense - TEHR-M - Temperature transmitter
{ S7_Optimized_Access := 'TRUE' }
AUTHOR : OlaBjornli
VERSION : 0.1
   VAR_INPUT
      mb_addr : USInt := 1;
   END_VAR
   VAR_OUTPUT
      temperature : Real;   // [Â°C]
      analogue_output : Real;   // [Â°F]
      potentiometer_position : Real;   // [%]
   END_VAR
   VAR_IN_OUT
      mb_query : "mb_query";
   END_VAR
   VAR
      sb : "mb_station_block_udt";
      read1 : Struct
         temperature : Int;   // [Â°C]
         analogue_output : Int;   // [Â°F]
         potentiometer_position : Int;   // [%]
      END_STRUCT;
   END_VAR
BEGIN
   // http://www.syxthsense.com/product/product_pdf/SN1.174-TEHR-M.pdf

   "mb_station_block_header"(sb := #sb, mb_query := #mb_query);

   #mb_query(mb_addr := #mb_addr,
             mode := #mb_query.c.mode.read,
             data_addr := 30001,
             data_ptr := #read1);
   #temperature := INT_TO_REAL(#read1.temperature) / 10;
   #analogue_output := INT_TO_REAL(#read1.analogue_output) / 10;
   #potentiometer_position := INT_TO_REAL(#read1.potentiometer_position) / 10;

   "mb_station_block_footer"(sb := #sb, mb_query := #mb_query);
END_FUNCTION_BLOCK

// folder: Library/Modbus/Station blocks/sb Untested/S/Scandinavian Electric

FUNCTION_BLOCK "Scandinavian_electric_CEM M-RS485"   // FB45, SCL
{ S7_Optimized_Access := 'TRUE' }
VERSION : 0.1
   VAR_INPUT
      mb_addr : UInt;
   END_VAR
   VAR_IN_OUT
      mb_query : "mb_query";
   END_VAR
   VAR
      sb : "mb_station_block_udt";
      read1 : Struct
         "Imported active energy" : UDInt;
         "Exported active energy" : UDInt;
         "Q1 Reactive energy" : UDInt;
         "Q2 Reactive energy" : UDInt;
         "Q3 Reactive energy" : UDInt;
         "Q4 Reactive energy" : UDInt;
      END_STRUCT;
      read2 : Struct
         "Partial imported active energy" : UDInt;
         "Partial exported active energy" : UDInt;
         "Q1 partial reactive energy" : UDInt;
         "Q2 partial reactive energy" : UDInt;
         "Q3 partial reactive energy" : UDInt;
         "Q4 partial reactive energy" : UDInt;
      END_STRUCT;
      serial_number : UDInt;
   END_VAR
BEGIN
   // Scandinavian Electric - Circutor - CEM M-RS485
   // Modbus interface for CEM energy meters

   // - Note: Only no parity.
   // - http://scel.no/produkter/energimaling_/_3_fase_malere/
   //   content/text_432575b2-b97f-4834-84d7-3fb83a2fdd40/1442214133237/
   //   cem_m_rs485.pdf
   // - (M014B01-03-14A)

   "mb_station_block_header"(sb := #sb, mb_query := #mb_query);
   #mb_query.mb_addr := #mb_addr;

   #mb_query.mode := #mb_query.c.read.holding_reg;
   #mb_query(data_addr := 16#0000, data_ptr := #read1);
   #mb_query(data_addr := 16#0030, data_ptr := #read2);
   #mb_query(data_addr := 16#2710, data_ptr := #serial_number);

   "mb_station_block_footer"(sb := #sb, mb_query := #mb_query);
END_FUNCTION_BLOCK

FUNCTION_BLOCK "Scandinavian_electric_Circutor_CBS"   // FB46, SCL
{ S7_Optimized_Access := 'TRUE' }
VERSION : 0.1
   VAR_INPUT
      mb_addr : UInt;
   END_VAR
   VAR_IN_OUT
      mb_query : "mb_query";
   END_VAR
   VAR
      sb : "mb_station_block_udt";
      data : Struct
         current : Array[1..8] of UInt;   // [mA]
         outputs : Array[1..8] of UInt;   // 0=Normal, 1=Pre-alarm, 2=Aktivert, 3=LÃ¥st
         pre_alarm_relay : UInt;
      END_STRUCT;
      limits : Array[1..8] of UInt;   // [mA]
   END_VAR
BEGIN
   // Scandinavian Electric - Circutor - CBS-8
   // 
   // - http://scel.no/produkter/jordfeilovervaking/
   //   varsler_panel_og_scanningsystem/content_2/
   //   text_8e3609e0-231d-4dfc-80a4-71ee43eee1af/1409662445698/cbs8.pdf

   "mb_station_block_header"(sb := #sb, mb_query := #mb_query);
   #mb_query.mb_addr := #mb_addr;

   #mb_query.mode := #mb_query.c.write.holding_reg;
   #mb_query(data_addr := 13, data_ptr := #limits);

   #mb_query.mode := #mb_query.c.read.holding_reg;
   #mb_query(data_addr := 2, data_ptr := #data);

   "mb_station_block_footer"(sb := #sb, mb_query := #mb_query);
END_FUNCTION_BLOCK

// folder: Library/Modbus/Station blocks/sb Untested/S/Schneider

FUNCTION_BLOCK "Schneider_ATV6xx"   // FB47, SCL
{ S7_Optimized_Access := 'TRUE' }
VERSION : 0.1
   VAR_INPUT
      mb_addr : USInt;
      ref_freq : Real;
   END_VAR
   VAR_IN_OUT
      mb_query : "mb_query";
   END_VAR
   VAR
      sb : "mb_station_block_udt";
      write1 : Struct
         cmd_reg : Struct
            x08_halt : Bool;
            x09 : Bool;
            x10 : Bool;
            x11_Reverse : Bool;
            x12 : Bool;
            x13 : Bool;
            x14 : Bool;
            x15 : Bool;
            x00_switch_on : Bool := TRUE;
            x01_enable_voltage : Bool := TRUE;
            x02_quick_stop : Bool;
            x03_Run : Bool;
            x04 : Bool;
            x05 : Bool;
            x06 : Bool;
            x07_fault_reset : Bool;
         END_STRUCT;
         ref_freq : Int;
      END_STRUCT;
      read1 : Struct
         status : Struct   // ETA
            x08 : Bool;
            x09_remote : Bool;   // Command or reference value via fieldbus
            x10_on_target : Bool;   // Reference value reached
            x11_ref_outside_lim : Bool;   // Reference value outside limits
            x12 : Bool;
            x13 : Bool;
            x14_stop_key : Bool;   // Manufacturer-specific Stop via STOP key
            x15_reverse : Bool;   // Manufacturer-specific
            x00_awaiting_power_stage_supply : Bool;
            x01_ready : Bool;
            x02_running : Bool;
            x03_fault : Bool;
            x04_power_stage_supply_present : Bool;
            x05_quick_stop : Bool;
            x06_power_stage_supply_disabled : Bool;
            x07_warning : Bool;
         END_STRUCT;
         output_frequency : Int;   // RFR
         frequency_reference_before_ramp : Int;   // FRH
         motor_current : Int;   // LCR
         motor_torque : Int;   // OTR
         ext_status_word : Word;
         mains_voltage : Int;   // ULN
         motor_voltage : Int;   // UOP
         drive_thermal_state : Int;   // THD
      END_STRUCT;
   END_VAR
BEGIN
   // Schneider - ATV6xx (EAV94279)
   //  
   // - http://www2.schneider-electric.com/resources/sites/SCHNEIDER_ELECTRIC/
   //   content/live/FAQS/275000/FA275868/en_US/
   //   Process%20drive%20communication%20parameters.xlsx
   // - https://profsector.com/media/catalogs/56e3af69500ef.pdf
   // - https://download.schneider-electric.com/
   //   files?p_enDocType=User+guide&p_File_Id=5470508810&
   //   p_File_Name=ATV600_EthernetIP_Modbus_TCP_Manual_EN_EAV6
   //   4328_02.pdf&p_Reference=EAV64328

   #write1.ref_freq := REAL_TO_INT(#ref_freq * 10);
   #write1.cmd_reg.x00_switch_on := #write1.cmd_reg.x03_Run := #ref_freq <> 0;

   "mb_station_block_header"(sb := #sb, mb_query := #mb_query);
   #mb_query.mb_addr := #mb_addr;

   #mb_query.mode := #mb_query.c.write.holding_reg;
   #mb_query(data_addr := 8501, data_ptr := #write1);

   #mb_query.mode := #mb_query.c.read.holding_reg;
   #mb_query(data_addr := 3201, data_ptr := #read1);

   "mb_station_block_footer"(sb := #sb, mb_query := #mb_query);
END_FUNCTION_BLOCK

FUNCTION_BLOCK "Schneider_SCADAPack_4000"   // FB51, SCL
{ S7_Optimized_Access := 'TRUE' }
VERSION : 0.1
   VAR_INPUT
      mb_addr : UInt;
   END_VAR
   VAR_IN_OUT
      mb_query : "mb_query";
   END_VAR
   VAR
      sb : "mb_station_block_udt";
      data : Array[1..3] of Int;
      setting : Array[1..3] of Int;
   END_VAR
BEGIN
   // Schneider - SCADAPack 4000 
   // Models 4012, 4032 and 4102 - Transmitters
   // 
   // Web: https://s3.amazonaws.com/cdn.freshdesk.com/data/helpdesk/
   // attachments/production/5013914262/original/
   // SCADAPack_4000_Series_Transmitters.pdf?
   // X-Amz-Algorithm=AWS4-HMAC-SHA256&X-Amz-Credential=
   // AKIAJ2JSYZ7O3I4JO6DA%2F20170919%2Fus-east-1%2Fs3%2Faws4_
   // request&X-Amz-Date=20170919T163931Z&X-Amz-Expires=300&X-Amz-
   // Signature=a206005821114e23f4a38162afdf9d14bd82209c246a378f18
   // 9af628740a1509&X-Amz-SignedHeaders=Host&response-content-type=
   // application%2Fpdf

   "mb_station_block_header"(sb := #sb, mb_query := #mb_query);
   #mb_query.mb_addr := #mb_addr;

   #mb_query.mode := #mb_query.c.mode.read;
   #mb_query(data_addr := 40116, data_ptr := #data);

   #mb_query.mode := #mb_query.c.mode.write;
   #mb_query(data_addr := 40060, data_ptr := #setting);

   "mb_station_block_footer"(sb := #sb, mb_query := #mb_query);

   (*
   Setting:

   value[1] and value[2]
   ------------------
   2 = Pascal (Pa)
   3 = kiloPascal (kPa)
   4 = megaPascal (MPa)
   5 = pounds per square inch (psi)
   6 = inches of water at 68 F
   7 = ftH2O
   8 = atm
   9 = bar
   10 = kg/cm2
   11 = g/cm2
   12 = cmHg
   13 = mmHg
   14 = torr
   15 = mH2O
   16 = cmH2O
   17 = mmH2O
   18 = inHg
   19 = mbar


   value[3]
   ------------------
   20 = degrees Celsius (ï‚°C)
   21 = degrees Fahrenheit (ï‚°F)
   22 = degrees Kelvin (K)
   23 = degrees Rankine(R)

   *)
END_FUNCTION_BLOCK

FUNCTION_BLOCK "Schneider_conzerv_EM6430"   // FB91, SCL
{ S7_Optimized_Access := 'TRUE' }
VERSION : 0.1
   VAR_INPUT
      mb_addr : USInt;
   END_VAR
   VAR_IN_OUT
      mb_query : "mb_query";
   END_VAR
   VAR
      sb : "mb_station_block_udt";
      read1_common : Struct
         Apparent_power_total : Real;
         Active_power_total : Real;
         Reactive_power_total : Real;
         Power_factor_average : Real;
         Voltage_average_phase_phase : Real;
         Voltage_average_phase_neutral : Real;
         Current_average : Real;
         Frequency : Real;   // Hz
      END_STRUCT;
      read2_phase : Array[1..3] of Struct
         Apparent_power : Real;
         Active_power : Real;
         Reactive_power : Real;
         Power_factor : Real;
         Voltage_phase_phase : Real;
         Voltage_phase_neutral : Real;
         Current : Real;
      END_STRUCT;
      read3_THD : Struct
         Voltage_THD : Array[1..3] of Real;
         Current_THD : Array[1..3] of Real;
      END_STRUCT;
      read4 : Struct
         Forward_apparent_energy : Real;
         Forward_active_energy : Real;
         Forward_reactive_inductive_energy : Real;
         Forward_reactive_capacitive_energy : Real;
         Reverse_apparent_energy : Real;
         Reverse_active_energy : Real;
         Reverse_reactive_inductive_Energy : Real;
         Reverse_reactive_capacitive_Energy : Real;
         Average_load_percentage : Real;
         Percentage_of_phase_load : Array[1..3] of Real;
         "Unbalanced_%load" : Real;
         "Unbalanced_%_voltage" : Real;
      END_STRUCT;
      read5_common_RMS : Struct
         Apparent_power_total : Real;
         Active_power_total : Real;
         Reactive_power_total : Real;
         Power_factor_average : Real;
         Voltage_average_phase_phase : Real;
         Voltage_average_phase_neutral : Real;
         Current_average : Real;
         Frequency : Real;   // Hz
         _ : UDInt;   // Reserved
         Number_of_interruption : UDInt;
      END_STRUCT;
   END_VAR
BEGIN
   // Schneider-electric - Conzerv EM6430 - Power meters
   // NHA12535-03
   // 
   // https://www.schneider-electric.com/resources/sites/SCHNEIDER_ELECTRIC/
   // content/live/FAQS/276000/FA276938/en_US/EM6430_User_Manual_NHA12535-03.pdf

   "mb_station_block_header"(sb := #sb, mb_query := #mb_query);
   #mb_query.mb_addr := #mb_addr; // Device address.

   #mb_query.mode := #mb_query.c.read.holding_reg;
   #mb_query(data_addr := 3901, data_ptr := #read1_common);
   #mb_query(data_addr := 3917, data_ptr := #read2_phase);
   #mb_query(data_addr := 3861, data_ptr := #read3_THD);
   #mb_query(data_addr := 3959, data_ptr := #read4);
   #mb_query(data_addr := 3001, data_ptr := #read5_common_RMS);

   "mb_station_block_footer"(sb := #sb, mb_query := #mb_query);
END_FUNCTION_BLOCK

// folder: Library/Modbus/Station blocks/sb Untested/S/Schneider/Altivar

FUNCTION_BLOCK "Schneider_Altivar_21"   // FB95, SCL
{ S7_Optimized_Access := 'TRUE' }
VERSION : 0.1
   VAR_INPUT
      mb_addr : UInt;
      ref : Real;
      acceleration_time : Real;
   END_VAR
   VAR_IN_OUT
      mb_query : "mb_query";
   END_VAR
   VAR
      sb : "mb_station_block_udt";
      data6 : Struct
         Output_current : Real;
         Voltage_DC_bus : Real;
         Output_frequency : Real;
      END_STRUCT;
      read1 : Struct   // 16#fd00
         Output_frequency : Word;
         stat : Struct
            x08 : Bool;
            x09_Reverse : Bool;
            x10_Run : Bool;
            x11_Coast_stop : Bool;
            x12_Emergency_stop : Bool;
            x13_Standby_ST_ON : Bool;   // Standby: Initialization completed, not failure stop status, not alarm stop status (MOFF, LL forced stop or forced stop due to a momentary power failure), ST=ON, and RUN=ON
            x14_Standby : Bool;   // Standby: Initialization completed, not failure stop status, and not alarm stop status (MOFF, LL forced stop or forced stop due to a momentary power failure)
            x15_Local : Bool;
            x00_Failure_FL : Bool;
            x01_Failure : Bool;
            x02_Alarm : Bool;
            x03_Main_circuit_undervoltage : Bool;
            x04_THR_2 : Bool;   // THR1: PT=set value, vL, vb, Thr - THR2: PT=0, F170, F172, F173
            x05_PI_control_OFF : Bool;
            x06_Acceleration2_deceleration2 : Bool;
            x07_DC_braking : Bool;
         END_STRUCT;
      END_STRUCT;
      read2 : Struct   // 16#fe45
         Command_mode : UInt;   // 0:Terminal board, 1:Operation panel, 2:Serial
         Setpoint_mode : UInt;   // 1 VIA, 2 VIB, 3 Operation panel, 4 Serial, 5 TB up down frequency, 255 Preset speed operation
      END_STRUCT;
      read3_alarm : Struct   // 16#fe91
         x08_Over_torque : Bool;
         x09_Cumulative_operation_hours : Bool;
         x10 : Bool;
         x11 : Bool;
         x12 : Bool;
         "x13_Main circuit_undervoltage" : Bool;   // same as MS-relay status
         x14_Decelerating_stopping : Bool;   // Related: F256 setting. At the time of the instant blackout, Forced deceleration/stop
         x15_Decelerating_stopping : Bool;   // Related: F302 setting. An automatic stop during the lower limit frequency continuance
         x00_Overcurrent : Bool;
         x01_Inverter_overload : Bool;
         x02_Motor_overload : Bool;
         x03_Overheat : Bool;
         x04_Overvoltage : Bool;
         x05_Main_circuit_undervoltage : Bool;
         x06 : Bool;
         x07_Undercurrent : Bool;
      END_STRUCT;
      read4_alarm2 : Struct   // 16#fe79
         x08 : Bool;
         x09 : Bool;
         x10 : Bool;
         x11 : Bool;
         x12 : Bool;
         x13 : Bool;
         x14 : Bool;
         x15 : Bool;
         x00_Fan_life_alarm : Bool;
         x01_Circuit_board_life : Bool;
         x02_Main_circuit_capacitor_life : Bool;
         x03_User_set_alarm : Bool;
         x04 : Bool;
         x05 : Bool;
         x06 : Bool;
         x07 : Bool;
      END_STRUCT;
      read5_trip_code : UInt;   // 16#fc90
      write1 : Struct
         cmd : Struct
            x08 : Bool;   // [08]
            reverse : Bool;   // [09]
            run : Bool;   // [10]
            coast_stop : Bool;   // [11]
            emergency_stop : Bool;   // [12]
            fault_reset : Bool;   // [13]
            setpoint_priority : Bool := TRUE;   // [14] Enabled regardless of the setting of FMOD
            command_priority : Bool := TRUE;   // [15] Enabled regardless of the setting of CMOD
            preset_speed_b0 : Bool;   // [00]
            preset_speed_b1 : Bool;   // [01]
            preset_speed_b2 : Bool;   // [02]
            x03 : Bool;   // [03]
            thr2 : Bool;   // [04] THR1 : PT=set value, vL, vb, tHr - THR2 : PT=0, F170, F172, F173
            PI_control : Bool;   // [05] 0:Normal operation, 1:PI OFF
            acceleration_deceleration_pattern_2 : Bool;   // [06] 0: Acceleration deceleration pattern 1
            DC_braking : Bool;   // [07]
         END_STRUCT;
         ref : UInt;
      END_STRUCT;
      write2_comm_fault_action : UInt;
      _ : Bool;
      sequence : "mb_sequence";
   END_VAR
   VAR_TEMP
      read6 : Struct   // 16#fe03
         Output_current : UInt;
         Voltage_DC_bus : UInt;
      END_STRUCT;
      u : UInt;
   END_VAR
BEGIN
   // Schneider (Telemecanique) - Altivar 21 inverter
   // VFD (AC-drive)

   (*
   Param:  Name:             Default:    Options:          
   F800    Baud rate         19200       0: 9600 bps, 1: 19200 bps     
   F801    Parity            Even        0: None, 1: Even, 2: Odd      
   F802    Modbus address    1           0 ... 247                     

   CMOD    2 -> Serial communication
   FMOD    4 -> Serial communication
   *)

   "mb_station_block_header"(sb := #sb, mb_query := #mb_query);
   #mb_query.mb_addr := #mb_addr;

   REGION Low priority queries     
       #sequence.conf.first_state := 1600;
       CASE "mb_sequence_init"(sequence := #sequence, mb_query := #mb_query) OF
               // ----- READ HOLDING REG ----- (State 3xx)
           300: // Where the drive take commands from: modbus or Terminal board.
               #mb_query(data_addr := 16#fe45, data_ptr := #read2); // 65093
           301: #mb_query(data_addr := 16#fe91, data_ptr := #read3_alarm);
           302: #mb_query(data_addr := 16#fe79, data_ptr := #read4_alarm2);
           303: #mb_query(data_addr := 16#fc90, data_ptr := #read5_trip_code);
           304: // Other data: Current, DC-bus
               #mb_query(data_addr := 16#fe03, data_ptr := #read6);
               IF #mb_query.Done THEN
                   #data6.Output_current := UINT_TO_REAL(#read6.Output_current) / 100;
                   #data6.Voltage_DC_bus := UINT_TO_REAL(#read6.Voltage_DC_bus) / 100;
               END_IF;
               #sequence.next_state := 1600;

               // ----- WRITE MULTIPLE HOLDING REG ----- (State 16xx)
           1600: // Behaviour on modbus fault
               #mb_query(data_addr := 16#f603, data_ptr := #write2_comm_fault_action);
           1601: // Acceleration time 1  (0.1)
               #u := REAL_TO_UINT(#acceleration_time * 10);
               #mb_query(data_addr := 16#f603, data_ptr := #u);
               #sequence.next_state := 300;
           ELSE
               #sequence.state += 1;
       END_CASE;
       #sequence(sb := #sb, mb_query := #mb_query);
   END_REGION

   REGION High priotiry querie   

       #write1.ref := REAL_TO_UINT(#ref * 100);
       #write1.cmd.run := #ref <> 0 AND #sequence.Done;
       #mb_query(mode := #mb_query.c.write.holding_reg, // 64000
                 data_addr := 16#fa00,
                 data_ptr := #write1);

       // Basic data, status word.
       #mb_query(mode := #mb_query.c.read.holding_reg,
                 data_addr := 16#fd00,
                 data_ptr := #read1); // 64768
       IF #mb_query.Done THEN
           #data6.Output_frequency :=
           (* *)UINT_TO_REAL(#read1.Output_frequency) / 100; // [%]
       END_IF;
   END_REGION

   "mb_station_block_footer"(sb := #sb, mb_query := #mb_query);

   (* Trip codes:
   NErr     0  0  No error
   OC1      1  1  Over-current during acceleration
   OC2      2  2  Over-current during deceleration
   OC3      3  3  Over-current during constant speed operation
   OCL      4  4  Over-current in load at startup
   OCA      5  5  Short circuit in arm
   EPHI     8  8  Input phase failure
   EPHO     9  9  Output phase failure
   OP1      A 10 Overvoltage during acceleration
   OP2      B 11 Overvoltage during deceleration
   OP3      C 12 Overvoltage during constant speed operation
   OL1      D 13 Over-LOAD in inverter
   OL2      E 14 Over-LOAD in motor
   OH      10 16 Overheat trip
   E       11 17 Emergency stop
   EEP1    12 18 EEPROM fault 1 (writing error)
   EEP2    13 19 EEPROM fault 2 (reading error)
   EEP3    14 20 EEPROM fault 3 (internal fault)
   Err2    15 21 RAM fault
   Err3    16 22 ROM fault
   Err4    17 23 CPU fault
   Err5    18 24 Communication error trip
   Err7    1A 26 Current detector fault
   Err8    1B 27 Optional circuit board type error
   UC      1D 29 Small-current trip
   UP1     1E 30 Trip due to undervoltage in main circuit
   Ot      20 32 Over-torque trip
   EF2     22 34 Ground fault trip (hardware detection)
   OC1P    25 37 Overcurrent flowing in element during acceleration
   OC2P    26 38 Overcurrent flowing in element during deceleration
   OC3P    27 39 Overcurrent flowing in element during operation
   EtYP    29 41 Inverter type error
   OH2     2E 46 External thermal input
   SOUt    2F 47 VIA cable break
   E-18    32 50 Break in an analog signal cable
   E-19    33 51 CPU fault
   E-20    34 52 Excess torque boost
   E-21    35 53 CPU fault
   Etn1    54 84 Auto-tuning error
   *)
END_FUNCTION_BLOCK

